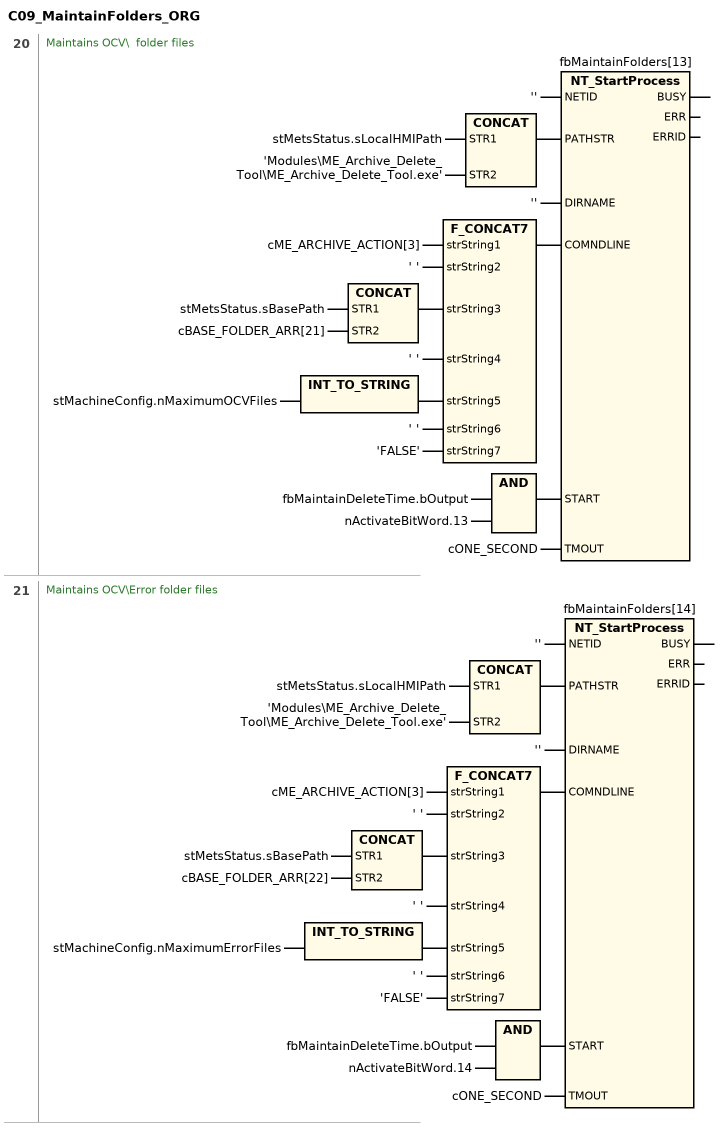
// NETWORK 20
// Maintains OCV\  folder files
fbMaintainFolders[13](
    NETID := '',
    PATHSTR := CONCAT(STR1 := stMetsStatus.sLocalHMIPath, STR2 := 'Modules\ME_Archive_Delete_Tool\ME_Archive_Delete_Tool.exe'),
    DIRNAME := '',
    COMNDLINE := F_CONCAT7(strString1 := cME_ARCHIVE_ACTION[3], strString2 := ' ', strString3 := CONCAT(STR1 := stMetsStatus.sBasePath, STR2 := cBASE_FOLDER_ARR[21]), strString4 := ' ', strString5 := INT_TO_STRING(stMachineConfig.nMaximumOCVFiles), strString6 := ' ', strString7 := 'FALSE'),
    START := fbMaintainDeleteTime.bOutput AND nActivateBitWord.13,
    TMOUT := cONE_SECOND); // NT_StartProcess

// NETWORK 21
// Maintains OCV\Error folder files
fbMaintainFolders[14](
    NETID := '',
    PATHSTR := CONCAT(STR1 := stMetsStatus.sLocalHMIPath, STR2 := 'Modules\ME_Archive_Delete_Tool\ME_Archive_Delete_Tool.exe'),
    DIRNAME := '',
    COMNDLINE := F_CONCAT7(strString1 := cME_ARCHIVE_ACTION[3], strString2 := ' ', strString3 := CONCAT(STR1 := stMetsStatus.sBasePath, STR2 := cBASE_FOLDER_ARR[22]), strString4 := ' ', strString5 := INT_TO_STRING(stMachineConfig.nMaximumErrorFiles), strString6 := ' ', strString7 := 'FALSE'),
    START := fbMaintainDeleteTime.bOutput AND nActivateBitWord.14,
    TMOUT := cONE_SECOND); // NT_StartProcess

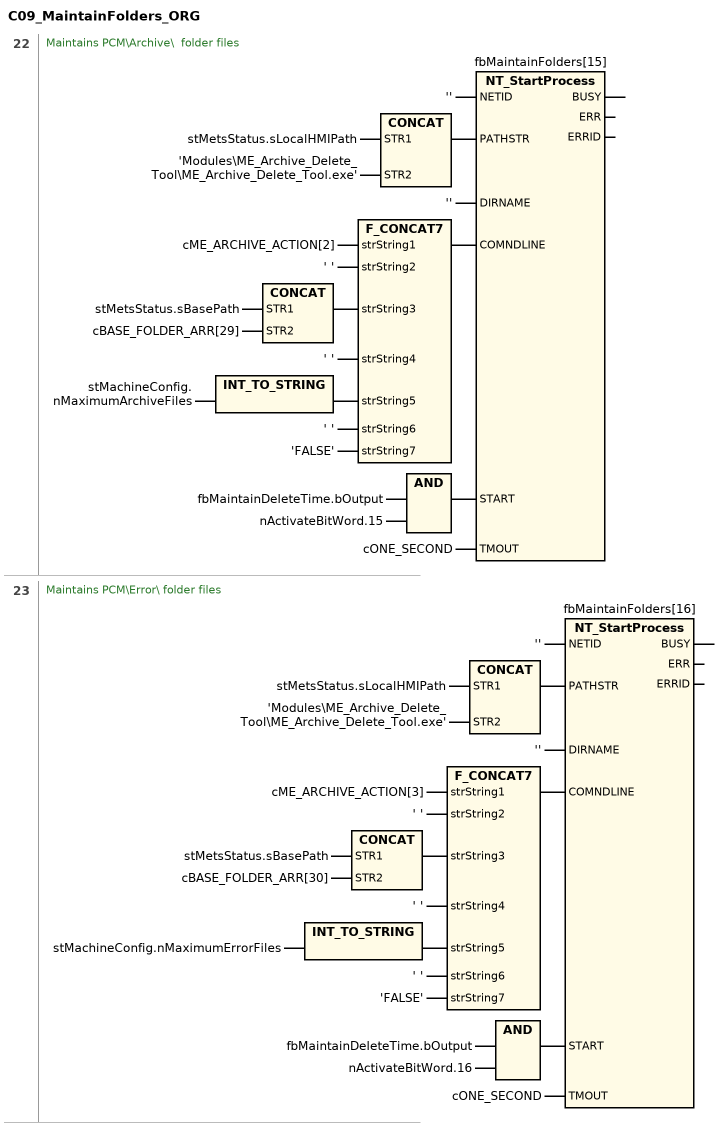
// NETWORK 22
// Maintains PCM\Archive\  folder files
fbMaintainFolders[15](
    NETID := '',
    PATHSTR := CONCAT(STR1 := stMetsStatus.sLocalHMIPath, STR2 := 'Modules\ME_Archive_Delete_Tool\ME_Archive_Delete_Tool.exe'),
    DIRNAME := '',
    COMNDLINE := F_CONCAT7(strString1 := cME_ARCHIVE_ACTION[2], strString2 := ' ', strString3 := CONCAT(STR1 := stMetsStatus.sBasePath, STR2 := cBASE_FOLDER_ARR[29]), strString4 := ' ', strString5 := INT_TO_STRING(stMachineConfig.nMaximumArchiveFiles), strString6 := ' ', strString7 := 'FALSE'),
    START := fbMaintainDeleteTime.bOutput AND nActivateBitWord.15,
    TMOUT := cONE_SECOND); // NT_StartProcess

// NETWORK 23
// Maintains PCM\Error\ folder files
fbMaintainFolders[16](
    NETID := '',
    PATHSTR := CONCAT(STR1 := stMetsStatus.sLocalHMIPath, STR2 := 'Modules\ME_Archive_Delete_Tool\ME_Archive_Delete_Tool.exe'),
    DIRNAME := '',
    COMNDLINE := F_CONCAT7(strString1 := cME_ARCHIVE_ACTION[3], strString2 := ' ', strString3 := CONCAT(STR1 := stMetsStatus.sBasePath, STR2 := cBASE_FOLDER_ARR[30]), strString4 := ' ', strString5 := INT_TO_STRING(stMachineConfig.nMaximumErrorFiles), strString6 := ' ', strString7 := 'FALSE'),
    START := fbMaintainDeleteTime.bOutput AND nActivateBitWord.16,
    TMOUT := cONE_SECOND); // NT_StartProcess

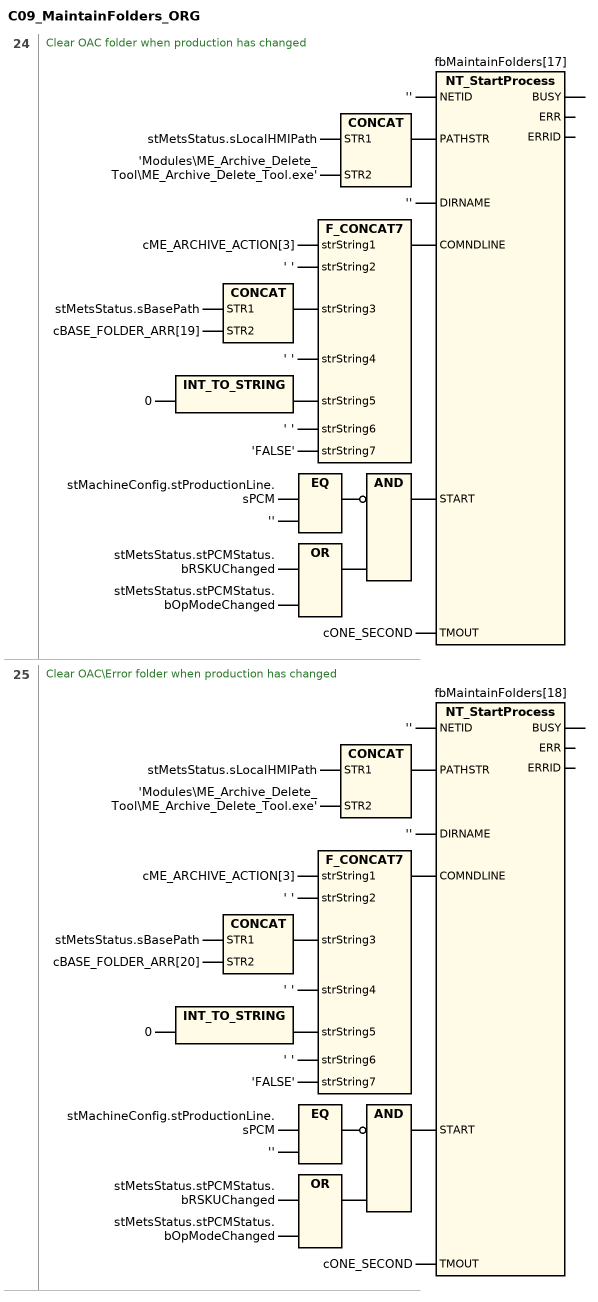
// NETWORK 24
// Clear OAC folder when production has changed
fbMaintainFolders[17](
    NETID := '',
    PATHSTR := CONCAT(STR1 := stMetsStatus.sLocalHMIPath, STR2 := 'Modules\ME_Archive_Delete_Tool\ME_Archive_Delete_Tool.exe'),
    DIRNAME := '',
    COMNDLINE := F_CONCAT7(strString1 := cME_ARCHIVE_ACTION[3], strString2 := ' ', strString3 := CONCAT(STR1 := stMetsStatus.sBasePath, STR2 := cBASE_FOLDER_ARR[19]), strString4 := ' ', strString5 := INT_TO_STRING(0), strString6 := ' ', strString7 := 'FALSE'),
    START := NOT (stMachineConfig.stProductionLine.sPCM = '') AND (stMetsStatus.stPCMStatus.bRSKUChanged OR stMetsStatus.stPCMStatus.bOpModeChanged),
    TMOUT := cONE_SECOND); // NT_StartProcess

// NETWORK 25
// Clear OAC\Error folder when production has changed
fbMaintainFolders[18](
    NETID := '',
    PATHSTR := CONCAT(STR1 := stMetsStatus.sLocalHMIPath, STR2 := 'Modules\ME_Archive_Delete_Tool\ME_Archive_Delete_Tool.exe'),
    DIRNAME := '',
    COMNDLINE := F_CONCAT7(strString1 := cME_ARCHIVE_ACTION[3], strString2 := ' ', strString3 := CONCAT(STR1 := stMetsStatus.sBasePath, STR2 := cBASE_FOLDER_ARR[20]), strString4 := ' ', strString5 := INT_TO_STRING(0), strString6 := ' ', strString7 := 'FALSE'),
    START := NOT (stMachineConfig.stProductionLine.sPCM = '') AND (stMetsStatus.stPCMStatus.bRSKUChanged OR stMetsStatus.stPCMStatus.bOpModeChanged),
    TMOUT := cONE_SECOND); // NT_StartProcess

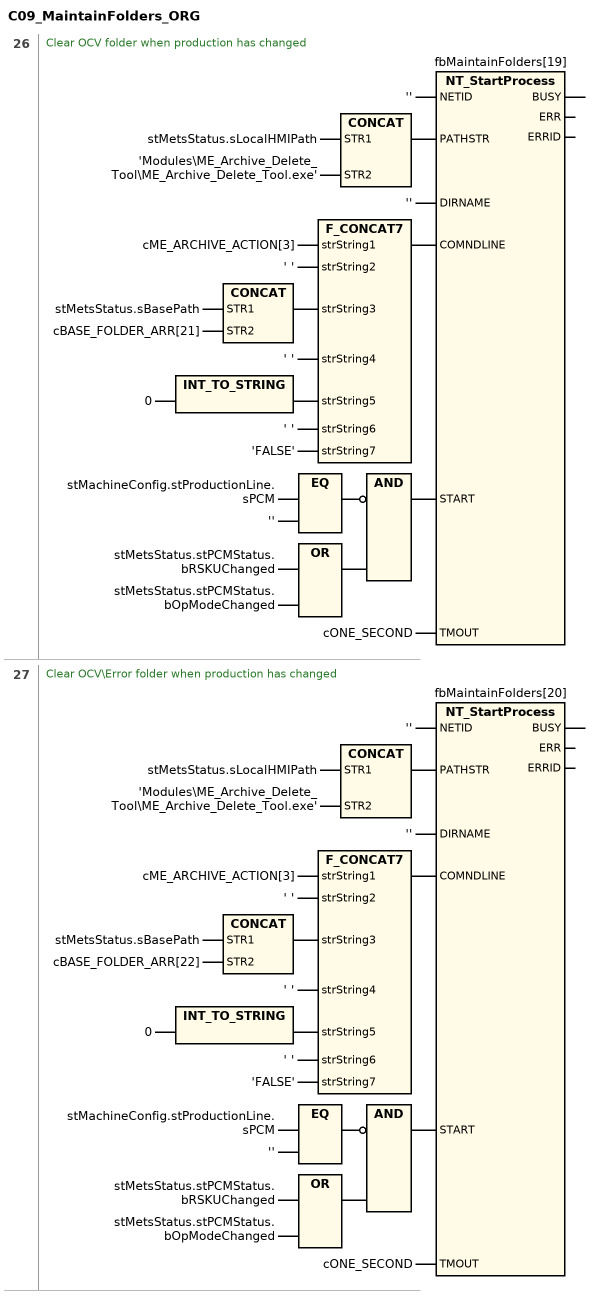
// NETWORK 26
// Clear OCV folder when production has changed
fbMaintainFolders[19](
    NETID := '',
    PATHSTR := CONCAT(STR1 := stMetsStatus.sLocalHMIPath, STR2 := 'Modules\ME_Archive_Delete_Tool\ME_Archive_Delete_Tool.exe'),
    DIRNAME := '',
    COMNDLINE := F_CONCAT7(strString1 := cME_ARCHIVE_ACTION[3], strString2 := ' ', strString3 := CONCAT(STR1 := stMetsStatus.sBasePath, STR2 := cBASE_FOLDER_ARR[21]), strString4 := ' ', strString5 := INT_TO_STRING(0), strString6 := ' ', strString7 := 'FALSE'),
    START := NOT (stMachineConfig.stProductionLine.sPCM = '') AND (stMetsStatus.stPCMStatus.bRSKUChanged OR stMetsStatus.stPCMStatus.bOpModeChanged),
    TMOUT := cONE_SECOND); // NT_StartProcess

// NETWORK 27
// Clear OCV\Error folder when production has changed
fbMaintainFolders[20](
    NETID := '',
    PATHSTR := CONCAT(STR1 := stMetsStatus.sLocalHMIPath, STR2 := 'Modules\ME_Archive_Delete_Tool\ME_Archive_Delete_Tool.exe'),
    DIRNAME := '',
    COMNDLINE := F_CONCAT7(strString1 := cME_ARCHIVE_ACTION[3], strString2 := ' ', strString3 := CONCAT(STR1 := stMetsStatus.sBasePath, STR2 := cBASE_FOLDER_ARR[22]), strString4 := ' ', strString5 := INT_TO_STRING(0), strString6 := ' ', strString7 := 'FALSE'),
    START := NOT (stMachineConfig.stProductionLine.sPCM = '') AND (stMetsStatus.stPCMStatus.bRSKUChanged OR stMetsStatus.stPCMStatus.bOpModeChanged),
    TMOUT := cONE_SECOND); // NT_StartProcess

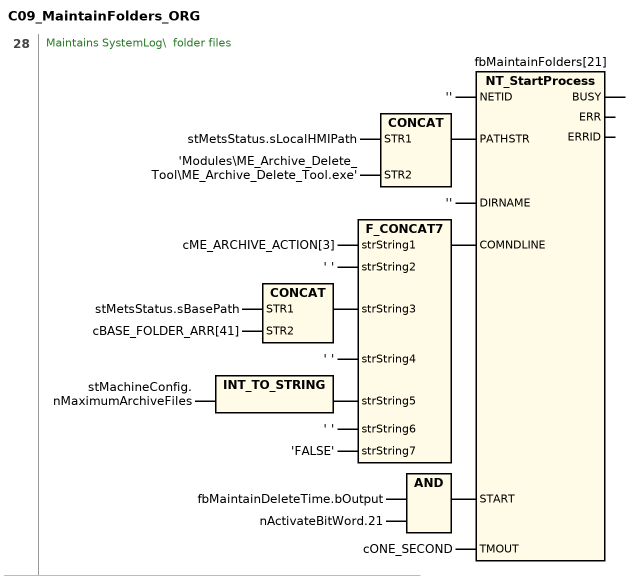
// NETWORK 28
// Maintains SystemLog\  folder files
fbMaintainFolders[21](
    NETID := '',
    PATHSTR := CONCAT(STR1 := stMetsStatus.sLocalHMIPath, STR2 := 'Modules\ME_Archive_Delete_Tool\ME_Archive_Delete_Tool.exe'),
    DIRNAME := '',
    COMNDLINE := F_CONCAT7(strString1 := cME_ARCHIVE_ACTION[3], strString2 := ' ', strString3 := CONCAT(STR1 := stMetsStatus.sBasePath, STR2 := cBASE_FOLDER_ARR[41]), strString4 := ' ', strString5 := INT_TO_STRING(stMachineConfig.nMaximumArchiveFiles), strString6 := ' ', strString7 := 'FALSE'),
    START := fbMaintainDeleteTime.bOutput AND nActivateBitWord.21,
    TMOUT := cONE_SECOND); // NT_StartProcess

ACTION ShiftActivationBit:
IF fbMaintainDeleteTime.bOutput	THEN
	IF nActivateBitWord = 0 THEN
		nActivateBitWord := 1;
	ELSE
		nActivateBitWord :=SHL(nActivateBitWord,1);
	END_IF
END_IF
END_ACTION

END_PROGRAM

// ---- POUs/_Exclude/F15_CaseControlCACData_ORG.TcPOU
PROGRAM F15_CaseControlCACData_ORG
VAR
	rtrigScanBarcode				: R_TRIG;
	fbScannerCtrl					: FB_SCANNER_CameraSelect;
	bScanCaseLabel				: BOOL;
	fbCaseLableEvaluation			: FB_SCANNER_Evaluation;

	rtrigSetCaseValidationOK			: R_TRIG;
	rtrigSetCaseValidationNOK		: R_TRIG;

	sCaseSerialCode				: T_CASE_Barcode;
	sFirstOuterInCase				: T_OUTER_Barcode;
	sLastOuterInCase				: T_OUTER_Barcode;
	sFirstPackSerialCode			: T_PACK_Barcode;
	sLastPackSerialCode				: T_PACK_Barcode;


	fbSequenceControl				: FB_SYSTEM_SeqControl;
	nSequenceStep				: INT;
	b00_Idle						: BOOL;
	b01_ScanLabel					: BOOL;
	b03_CreateFileName			: BOOL;
	b05_MoveCaseData				: BOOL;
	b08_WriteFSSFile				: BOOL;
	b10_CaseTraceValid			: BOOL;
	b18_CaseValid					: BOOL;
	b19_CaseInvalid				: BOOL;
	b20_Done						: BOOL;

	bDone						: BOOL;
	bBusy						: BOOL;
	tonScanTimeout					: TON;
	tonOverTime				: TON;

	rtrigCACData				: R_TRIG;
	tF15TimeExecution		: TIME;
	bTestSeq						: BOOL;
	sCACFileTemplate				: T_CAC_Filename;

	stValidateCACData				: ST_CAC_Data;
	fbMoveCaseData				: FB_CASE_ValidateAndMoveCACData;

	sPrintCaseContent				: STRING(255);

	fbPopulateCHMData				: FB_CHM_PopulateDataForFSS3;
	fbWriteCHMFile				: FB_CHM_WriteFSS3Files; (*Old system supporting FSS2 -> FB_CHM_WriteFSSFile;*)

	fbWriteCACToArchive 			: FB_CAC_WriteToArchive_v2;
	fbWriteCACToArchiveDB			: FB_CAC_WriteHierachyToDB;
	fbCaseStatusPulse				: TON;
	bCACValid					: BOOL;
	bCHMValid					: BOOL;


	fbMoveVerifiedCAC				: FB_CASE_MoveVerifiedCAC;
	fbMoveFailedCAC				: FB_CASE_MoveFailedCAC;

	fbCaseEfficiency				: FB_KPI_GenericEfficiency;
	fbCaseInspectionEfficiency		: FB_KPI_CaseEfficiency;
	(*fbCaseInspectionEfficiency		: FB_KPI_PACAN_CaseEfficiency;*)
	fbRejectCount					: CTU;
	nRejectActualCount				: INT;

	fbCaseValidationScanned			: FB_CTU32;
	fbCaseValidationCorrect			: FB_CTU32;
	fbCaseValidationNoCaseLabel		: FB_CTU32;
	fbCaseValidationCasePackerReject	: FB_CTU32;

	aLastCaseBarcodes				: ARRAY[1..cMAX_LAST_CASE_BARCODES] OF T_CASE_Barcode;
	fbAddVerifiedCaseBarcode		: FB_CASE_AddVerifiedCaseBarcode;

	fbCaseLevelCounter	: FB_KPI_CaseLevelCounter;
	tofCaseValidationCameraOFFDelay 	: TOF;

	fbFileWriteCACError				: FB_LOG_FileWriteError;
	fbFileWriteCHMError			: FB_LOG_FileWriteError;

END_VAR
(*
VAR CONSTANT
	sOptions						: ST_SCANNER_Options := (eScannerType := E_MV_440SR_FULL, nImageBuffer := 1, nExpectedResp := 1);
END_VAR*)
VAR // added by the converter: edge detectors and wires of the graphical bodies
    _w1 : ANY;
    _w2, _w3 : BOOL;
END_VAR

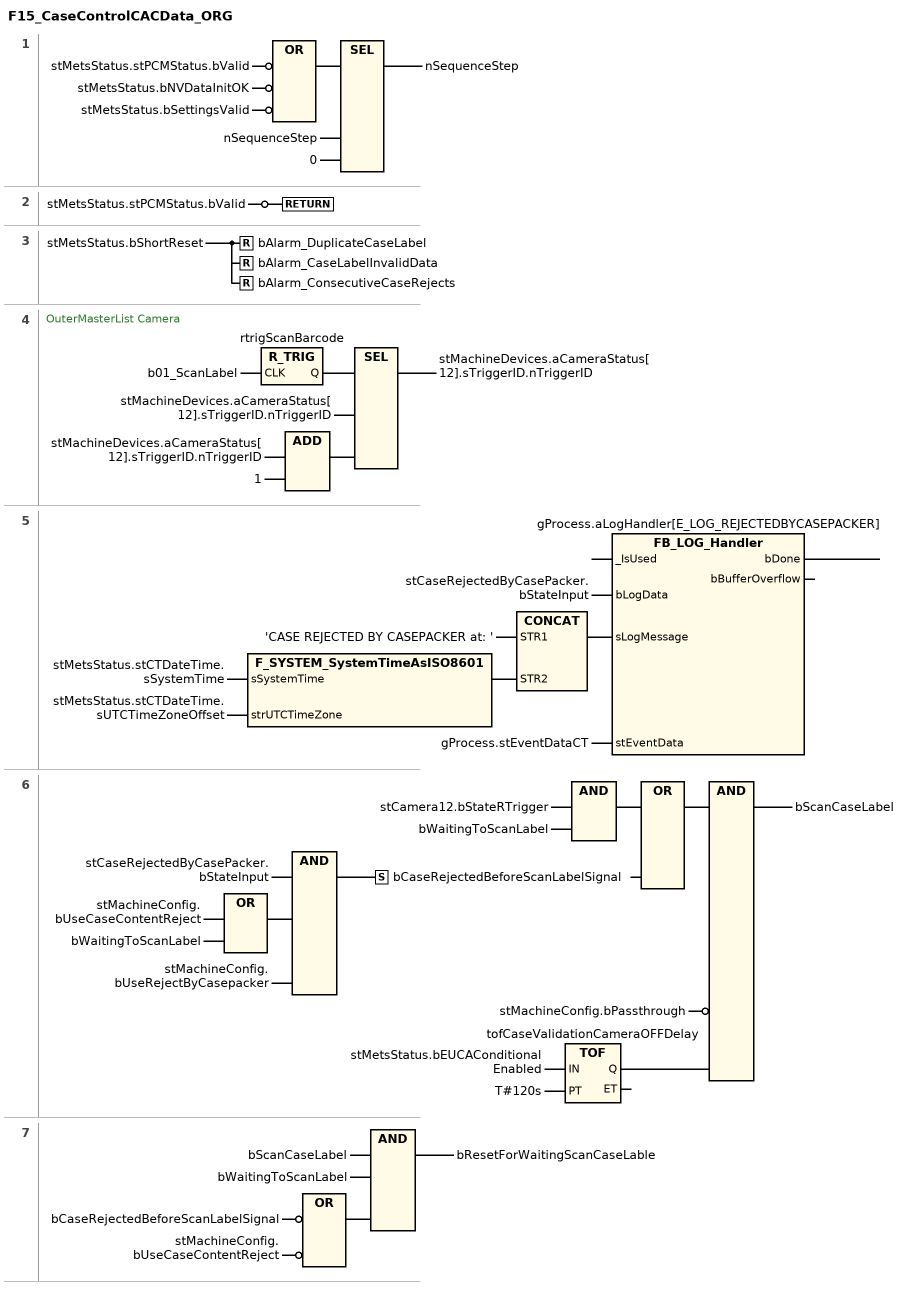
// NETWORK 1
nSequenceStep := SEL(NOT stMetsStatus.stPCMStatus.bValid OR NOT stMetsStatus.bNVDataInitOK OR NOT stMetsStatus.bSettingsValid, nSequenceStep, 0);

// NETWORK 2
IF NOT stMetsStatus.stPCMStatus.bValid THEN RETURN; END_IF

// NETWORK 3
bAlarm_DuplicateCaseLabel R= stMetsStatus.bShortReset;
bAlarm_CaseLabelInvalidData R= stMetsStatus.bShortReset;
bAlarm_ConsecutiveCaseRejects R= stMetsStatus.bShortReset;

// NETWORK 4
// OuterMasterList Camera
rtrigScanBarcode(CLK := b01_ScanLabel); // R_TRIG
stMachineDevices.aCameraStatus[12].sTriggerID.nTriggerID := SEL(rtrigScanBarcode.Q, stMachineDevices.aCameraStatus[12].sTriggerID.nTriggerID, stMachineDevices.aCameraStatus[12].sTriggerID.nTriggerID + 1);

// NETWORK 5
gProcess.aLogHandler[E_LOG_REJECTEDBYCASEPACKER](
    bLogData := stCaseRejectedByCasePacker.bStateInput,
    sLogMessage := CONCAT(STR1 := 'CASE REJECTED BY CASEPACKER at: ', STR2 := F_SYSTEM_SystemTimeAsISO8601(sSystemTime := stMetsStatus.stCTDateTime.sSystemTime, strUTCTimeZone := stMetsStatus.stCTDateTime.sUTCTimeZoneOffset)),
    stEventData := gProcess.stEventDataCT); // FB_LOG_Handler

// NETWORK 6
_w1 := stCaseRejectedByCasePacker.bStateInput AND (stMachineConfig.bUseCaseContentReject OR bWaitingToScanLabel) AND stMachineConfig.bUseRejectByCasepacker;
bCaseRejectedBeforeScanLabelSignal S= _w1;
tofCaseValidationCameraOFFDelay(IN := stMetsStatus.bEUCAConditionalEnabled, PT := T#120s); // TOF
bScanCaseLabel := (stCamera12.bStateRTrigger AND bWaitingToScanLabel OR _w1) AND NOT stMachineConfig.bPassthrough AND tofCaseValidationCameraOFFDelay.Q;

// NETWORK 7
bResetForWaitingScanCaseLable := bScanCaseLabel AND bWaitingToScanLabel AND (NOT bCaseRejectedBeforeScanLabelSignal OR NOT stMachineConfig.bUseCaseContentReject);

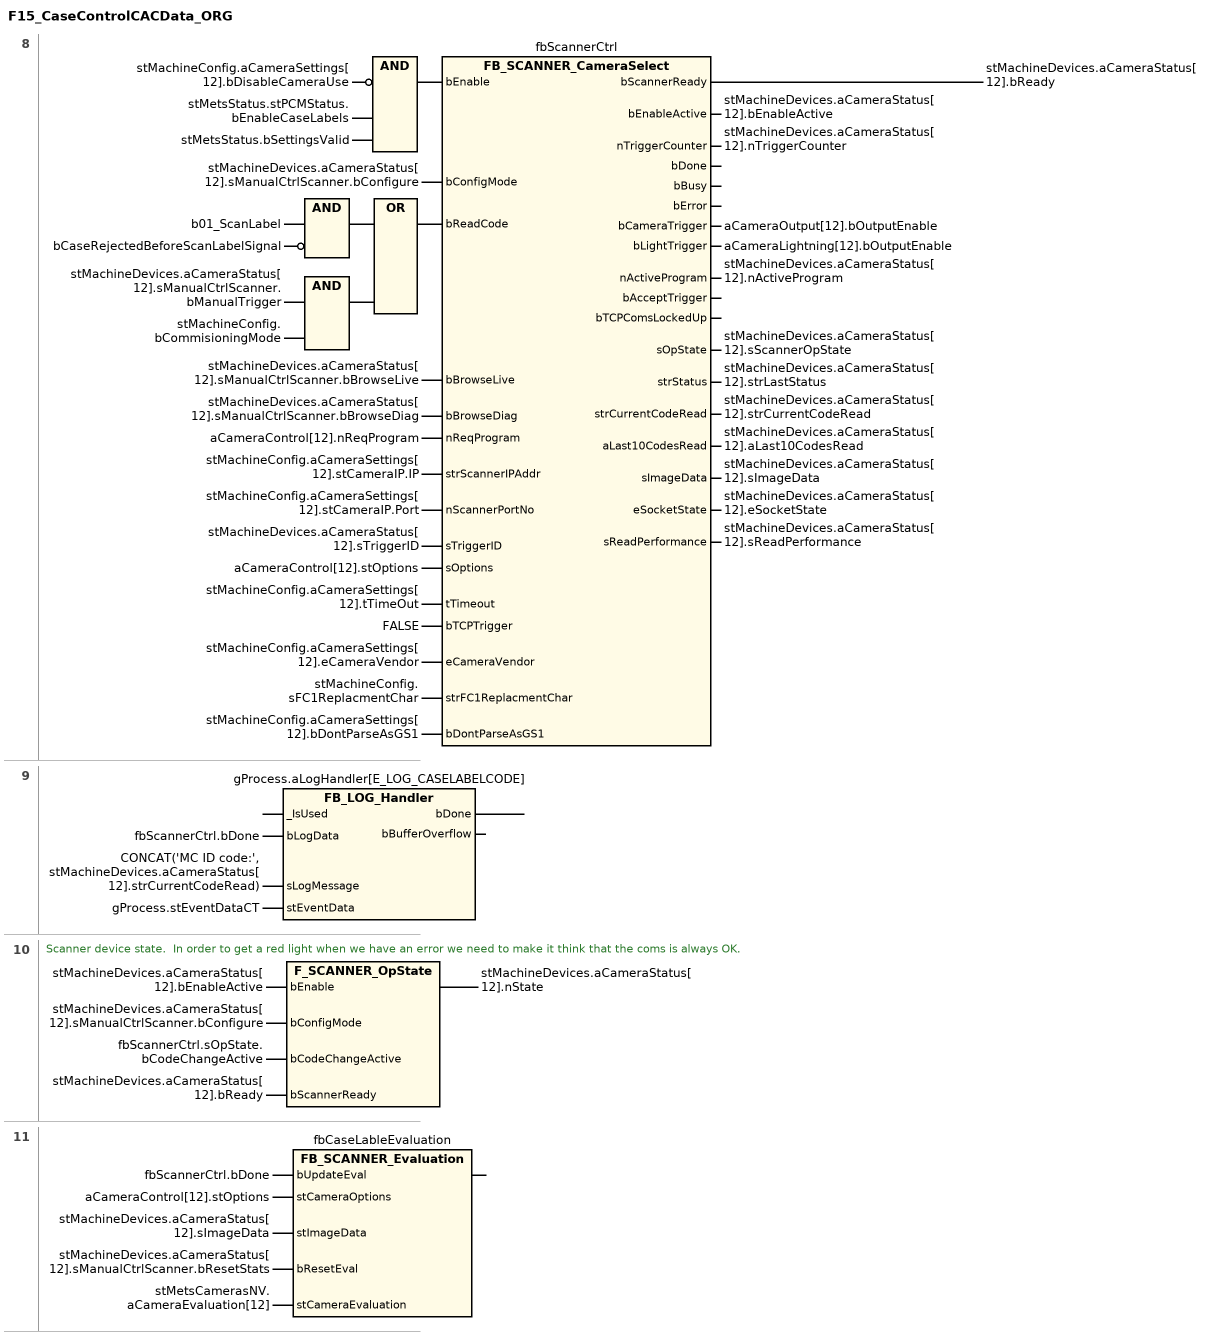
// NETWORK 8
fbScannerCtrl(
    bEnable := NOT stMachineConfig.aCameraSettings[12].bDisableCameraUse AND stMetsStatus.stPCMStatus.bEnableCaseLabels AND stMetsStatus.bSettingsValid,
    bConfigMode := stMachineDevices.aCameraStatus[12].sManualCtrlScanner.bConfigure,
    bReadCode := b01_ScanLabel AND NOT bCaseRejectedBeforeScanLabelSignal OR stMachineDevices.aCameraStatus[12].sManualCtrlScanner.bManualTrigger AND stMachineConfig.bCommisioningMode,
    bBrowseLive := stMachineDevices.aCameraStatus[12].sManualCtrlScanner.bBrowseLive,
    bBrowseDiag := stMachineDevices.aCameraStatus[12].sManualCtrlScanner.bBrowseDiag,
    nReqProgram := aCameraControl[12].nReqProgram,
    strScannerIPAddr := stMachineConfig.aCameraSettings[12].stCameraIP.IP,
    nScannerPortNo := stMachineConfig.aCameraSettings[12].stCameraIP.Port,
    sTriggerID := stMachineDevices.aCameraStatus[12].sTriggerID,
    sOptions := aCameraControl[12].stOptions,
    tTimeout := stMachineConfig.aCameraSettings[12].tTimeOut,
    bTCPTrigger := FALSE,
    eCameraVendor := stMachineConfig.aCameraSettings[12].eCameraVendor,
    strFC1ReplacmentChar := stMachineConfig.sFC1ReplacmentChar,
    bDontParseAsGS1 := stMachineConfig.aCameraSettings[12].bDontParseAsGS1,
    bEnableActive => stMachineDevices.aCameraStatus[12].bEnableActive,
    nTriggerCounter => stMachineDevices.aCameraStatus[12].nTriggerCounter,
    bCameraTrigger => aCameraOutput[12].bOutputEnable,
    bLightTrigger => aCameraLightning[12].bOutputEnable,
    nActiveProgram => stMachineDevices.aCameraStatus[12].nActiveProgram,
    sOpState => stMachineDevices.aCameraStatus[12].sScannerOpState,
    strStatus => stMachineDevices.aCameraStatus[12].strLastStatus,
    strCurrentCodeRead => stMachineDevices.aCameraStatus[12].strCurrentCodeRead,
    aLast10CodesRead => stMachineDevices.aCameraStatus[12].aLast10CodesRead,
    sImageData => stMachineDevices.aCameraStatus[12].sImageData,
    eSocketState => stMachineDevices.aCameraStatus[12].eSocketState,
    sReadPerformance => stMachineDevices.aCameraStatus[12].sReadPerformance); // FB_SCANNER_CameraSelect
stMachineDevices.aCameraStatus[12].bReady := fbScannerCtrl.bScannerReady;

// NETWORK 9
gProcess.aLogHandler[E_LOG_CASELABELCODE](
    bLogData := fbScannerCtrl.bDone,
    sLogMessage := CONCAT('MC ID code:', stMachineDevices.aCameraStatus[12].strCurrentCodeRead),
    stEventData := gProcess.stEventDataCT); // FB_LOG_Handler

// NETWORK 10
// Scanner device state.  In order to get a red light when we have an error we need to make it think that the coms is always OK.
stMachineDevices.aCameraStatus[12].nState := F_SCANNER_OpState(bEnable := stMachineDevices.aCameraStatus[12].bEnableActive, bConfigMode := stMachineDevices.aCameraStatus[12].sManualCtrlScanner.bConfigure, bCodeChangeActive := fbScannerCtrl.sOpState.bCodeChangeActive, bScannerReady := stMachineDevices.aCameraStatus[12].bReady);

// NETWORK 11
fbCaseLableEvaluation(
    bUpdateEval := fbScannerCtrl.bDone,
    stCameraOptions := aCameraControl[12].stOptions,
    stImageData := stMachineDevices.aCameraStatus[12].sImageData,
    bResetEval := stMachineDevices.aCameraStatus[12].sManualCtrlScanner.bResetStats,
    stCameraEvaluation := stMetsCamerasNV.aCameraEvaluation[12]); // FB_SCANNER_Evaluation

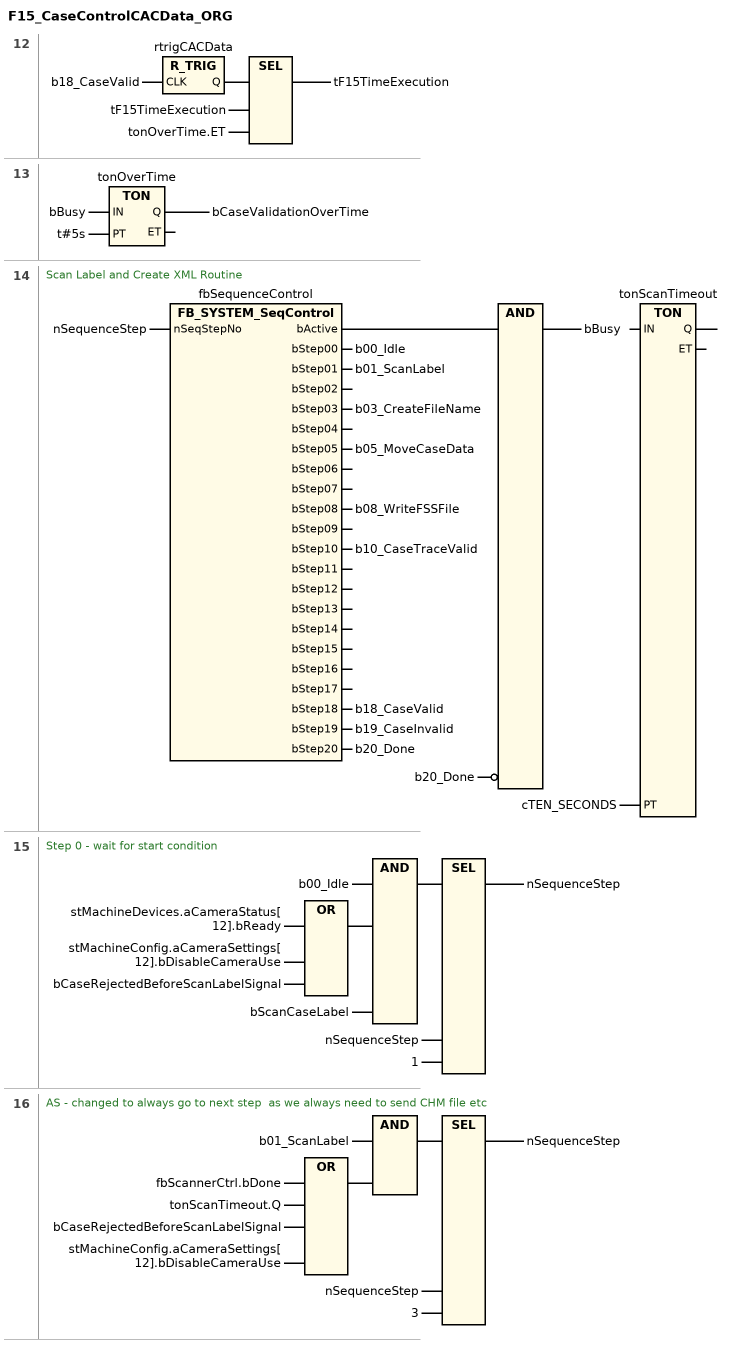
// NETWORK 12
rtrigCACData(CLK := b18_CaseValid); // R_TRIG
tF15TimeExecution := SEL(rtrigCACData.Q, tF15TimeExecution, tonOverTime.ET);

// NETWORK 13
tonOverTime(IN := bBusy, PT := t#5s); // TON
bCaseValidationOverTime := tonOverTime.Q;

// NETWORK 14
// 					Scan Label and Create XML Routine
//
//
//
fbSequenceControl(
    nSeqStepNo := nSequenceStep,
    bStep00 => b00_Idle,
    bStep01 => b01_ScanLabel,
    bStep03 => b03_CreateFileName,
    bStep05 => b05_MoveCaseData,
    bStep08 => b08_WriteFSSFile,
    bStep10 => b10_CaseTraceValid,
    bStep18 => b18_CaseValid,
    bStep19 => b19_CaseInvalid,
    bStep20 => b20_Done); // FB_SYSTEM_SeqControl
_w2 := fbSequenceControl.bActive AND NOT b20_Done;
bBusy := _w2;
tonScanTimeout(IN := _w2, PT := cTEN_SECONDS); // TON

// NETWORK 15
// 					Step 0 - wait for start condition
//
//
nSequenceStep := SEL(b00_Idle AND (stMachineDevices.aCameraStatus[12].bReady OR stMachineConfig.aCameraSettings[12].bDisableCameraUse OR bCaseRejectedBeforeScanLabelSignal) AND bScanCaseLabel, nSequenceStep, 1);

// NETWORK 16
// 					AS - changed to always go to next step  as we always need to send CHM file etc
//
//
nSequenceStep := SEL(b01_ScanLabel AND (fbScannerCtrl.bDone OR tonScanTimeout.Q OR bCaseRejectedBeforeScanLabelSignal OR stMachineConfig.aCameraSettings[12].bDisableCameraUse), nSequenceStep, 3);

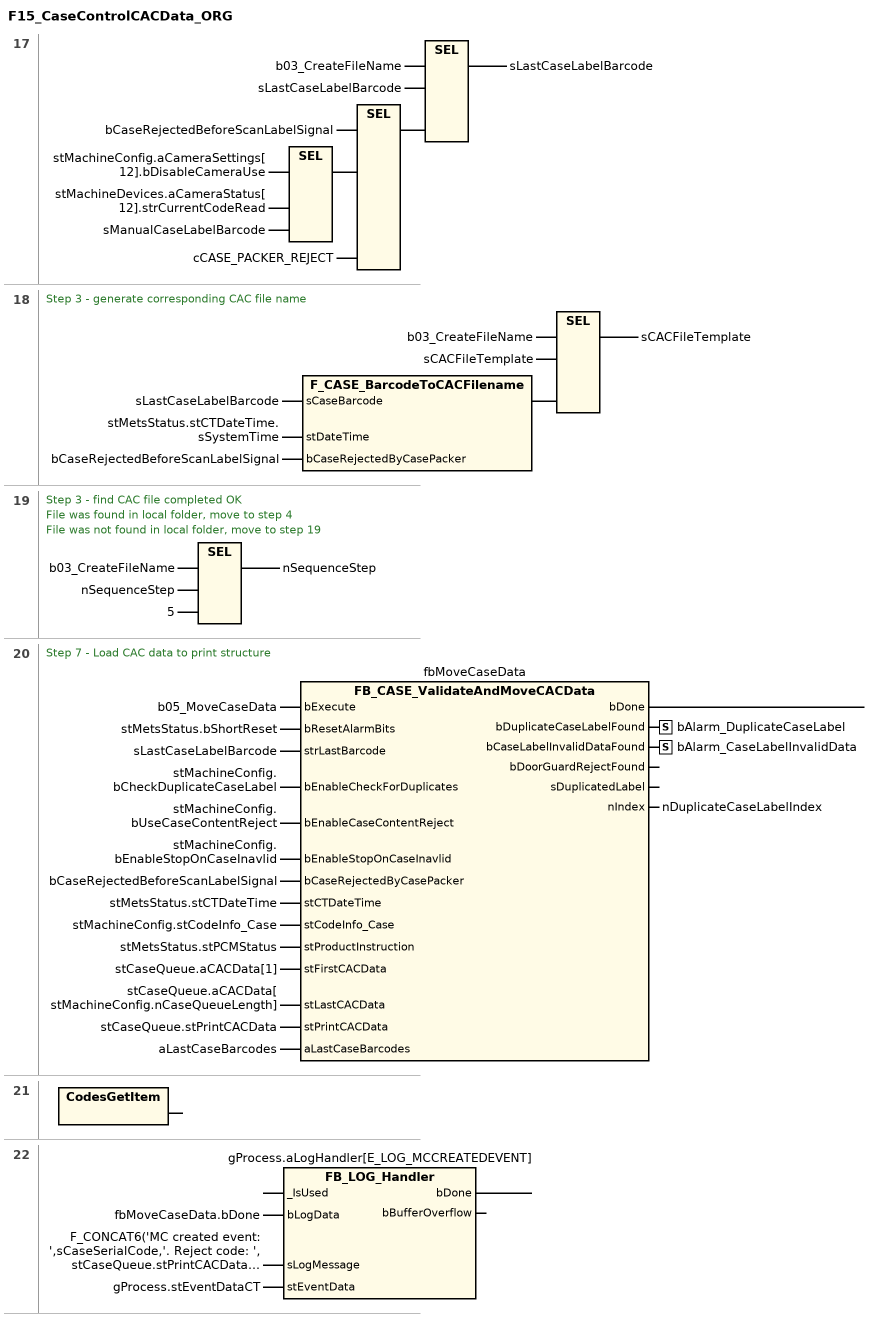
// NETWORK 17
sLastCaseLabelBarcode := SEL(b03_CreateFileName, sLastCaseLabelBarcode, SEL(bCaseRejectedBeforeScanLabelSignal, SEL(stMachineConfig.aCameraSettings[12].bDisableCameraUse, stMachineDevices.aCameraStatus[12].strCurrentCodeRead, sManualCaseLabelBarcode), cCASE_PACKER_REJECT));

// NETWORK 18
// Step 3 - generate corresponding CAC file name
sCACFileTemplate := SEL(b03_CreateFileName, sCACFileTemplate, F_CASE_BarcodeToCACFilename(sCaseBarcode := sLastCaseLabelBarcode, stDateTime := stMetsStatus.stCTDateTime.sSystemTime, bCaseRejectedByCasePacker := bCaseRejectedBeforeScanLabelSignal));

// NETWORK 19
// 					Step 3 - find CAC file completed OK
// File was found in local folder, move to step 4
// File was not found in local folder, move to step 19
//
nSequenceStep := SEL(b03_CreateFileName, nSequenceStep, 5);

// NETWORK 20
// Step 7 - Load CAC data to print structure
fbMoveCaseData(
    bExecute := b05_MoveCaseData,
    bResetAlarmBits := stMetsStatus.bShortReset,
    strLastBarcode := sLastCaseLabelBarcode,
    bEnableCheckForDuplicates := stMachineConfig.bCheckDuplicateCaseLabel,
    bEnableCaseContentReject := stMachineConfig.bUseCaseContentReject,
    bEnableStopOnCaseInavlid := stMachineConfig.bEnableStopOnCaseInavlid,
    bCaseRejectedByCasePacker := bCaseRejectedBeforeScanLabelSignal,
    stCTDateTime := stMetsStatus.stCTDateTime,
    stCodeInfo_Case := stMachineConfig.stCodeInfo_Case,
    stProductInstruction := stMetsStatus.stPCMStatus,
    stFirstCACData := stCaseQueue.aCACData[1],
    stLastCACData := stCaseQueue.aCACData[stMachineConfig.nCaseQueueLength],
    stPrintCACData := stCaseQueue.stPrintCACData,
    aLastCaseBarcodes := aLastCaseBarcodes,
    nIndex => nDuplicateCaseLabelIndex); // FB_CASE_ValidateAndMoveCACData
bAlarm_DuplicateCaseLabel S= fbMoveCaseData.bDuplicateCaseLabelFound;
bAlarm_CaseLabelInvalidData S= fbMoveCaseData.bCaseLabelInvalidDataFound;

// NETWORK 21
CodesGetItem();

// NETWORK 22
gProcess.aLogHandler[E_LOG_MCCREATEDEVENT](
    bLogData := fbMoveCaseData.bDone,
    sLogMessage := F_CONCAT6('MC created event: ',sCaseSerialCode,'. Reject code: ', stCaseQueue.stPrintCACData.CaseRejectCode,', with case content: ', sPrintCaseContent),
    stEventData := gProcess.stEventDataCT); // FB_LOG_Handler

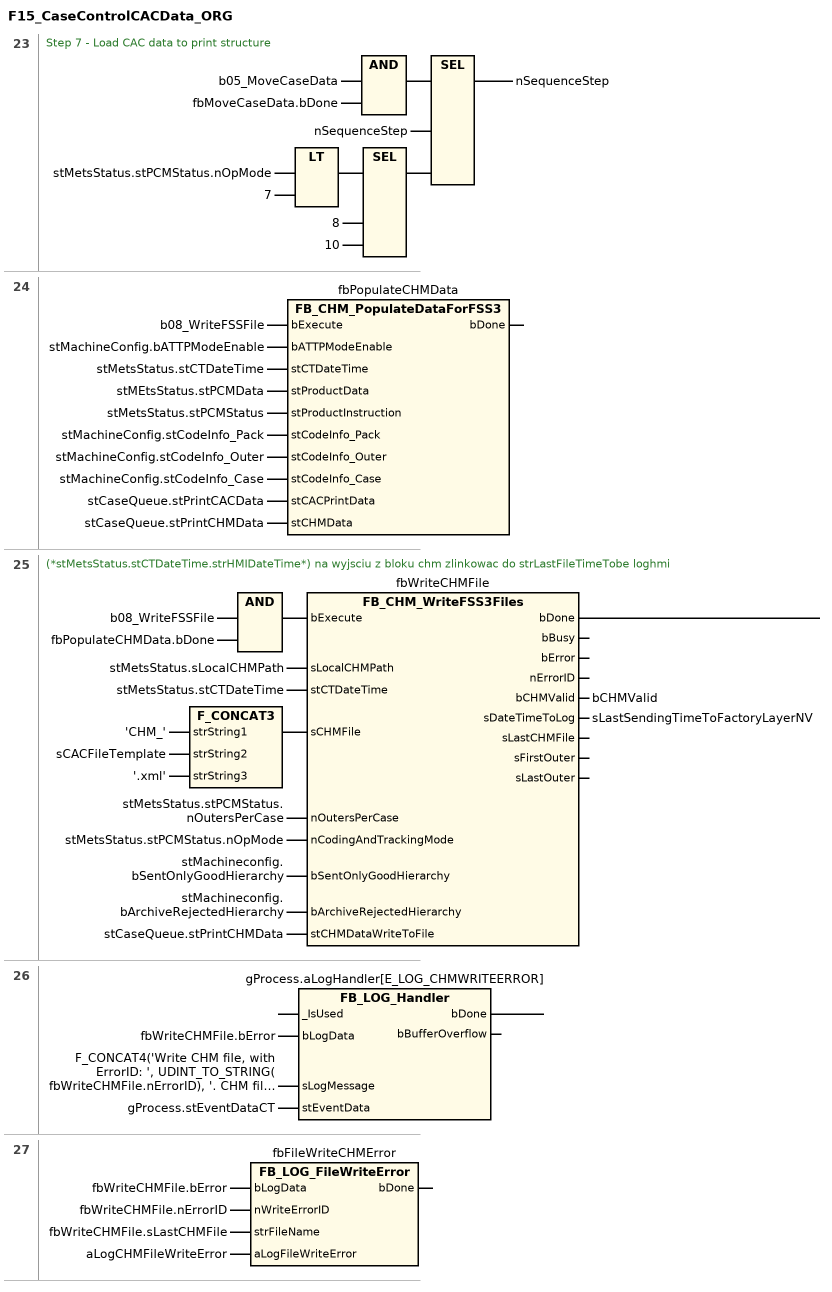
// NETWORK 23
// 					Step 7 - Load CAC data to print structure
//
//
nSequenceStep := SEL(b05_MoveCaseData AND fbMoveCaseData.bDone, nSequenceStep, SEL(stMetsStatus.stPCMStatus.nOpMode < 7, 8, 10));

// NETWORK 24
fbPopulateCHMData(
    bExecute := b08_WriteFSSFile,
    bATTPModeEnable := stMachineConfig.bATTPModeEnable,
    stCTDateTime := stMetsStatus.stCTDateTime,
    stProductData := stMEtsStatus.stPCMData,
    stProductInstruction := stMetsStatus.stPCMStatus,
    stCodeInfo_Pack := stMachineConfig.stCodeInfo_Pack,
    stCodeInfo_Outer := stMachineConfig.stCodeInfo_Outer,
    stCodeInfo_Case := stMachineConfig.stCodeInfo_Case,
    stCACPrintData := stCaseQueue.stPrintCACData,
    stCHMData := stCaseQueue.stPrintCHMData); // FB_CHM_PopulateDataForFSS3

// NETWORK 25
// (*stMetsStatus.stCTDateTime.strHMIDateTime*) na wyjsciu z bloku chm zlinkowac do strLastFileTimeTobe loghmi
fbWriteCHMFile(
    bExecute := b08_WriteFSSFile AND fbPopulateCHMData.bDone,
    sLocalCHMPath := stMetsStatus.sLocalCHMPath,
    stCTDateTime := stMetsStatus.stCTDateTime,
    sCHMFile := F_CONCAT3(strString1 := 'CHM_', strString2 := sCACFileTemplate, strString3 := '.xml'),
    nOutersPerCase := stMetsStatus.stPCMStatus.nOutersPerCase,
    nCodingAndTrackingMode := stMetsStatus.stPCMStatus.nOpMode,
    bSentOnlyGoodHierarchy := stMachineconfig.bSentOnlyGoodHierarchy,
    bArchiveRejectedHierarchy := stMachineconfig.bArchiveRejectedHierarchy,
    stCHMDataWriteToFile := stCaseQueue.stPrintCHMData,
    bCHMValid => bCHMValid,
    sDateTimeToLog => sLastSendingTimeToFactoryLayerNV); // FB_CHM_WriteFSS3Files

// NETWORK 26
gProcess.aLogHandler[E_LOG_CHMWRITEERROR](
    bLogData := fbWriteCHMFile.bError,
    sLogMessage := F_CONCAT4('Write CHM file, with ErrorID: ', UDINT_TO_STRING(fbWriteCHMFile.nErrorID), '. CHM file name: ', fbWriteCHMFile.sCHMFile),
    stEventData := gProcess.stEventDataCT); // FB_LOG_Handler

// NETWORK 27
fbFileWriteCHMError(
    bLogData := fbWriteCHMFile.bError,
    nWriteErrorID := fbWriteCHMFile.nErrorID,
    strFileName := fbWriteCHMFile.sLastCHMFile,
    aLogFileWriteError := aLogCHMFileWriteError); // FB_LOG_FileWriteError

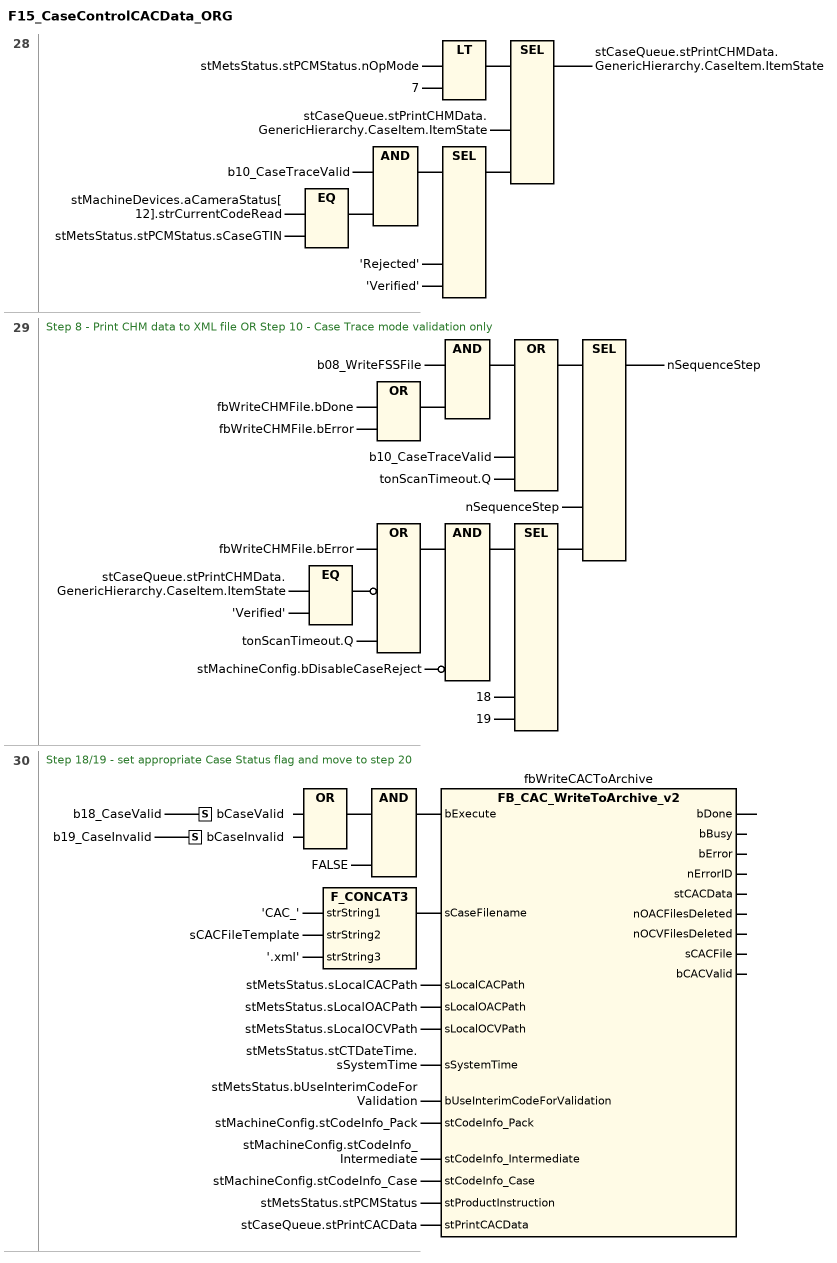
// NETWORK 28
stCaseQueue.stPrintCHMData.GenericHierarchy.CaseItem.ItemState := SEL(stMetsStatus.stPCMStatus.nOpMode < 7, stCaseQueue.stPrintCHMData.GenericHierarchy.CaseItem.ItemState, SEL(b10_CaseTraceValid AND stMachineDevices.aCameraStatus[12].strCurrentCodeRead = stMetsStatus.stPCMStatus.sCaseGTIN, 'Rejected', 'Verified'));

// NETWORK 29
// Step 8 - Print CHM data to XML file OR Step 10 - Case Trace mode validation only
nSequenceStep := SEL(b08_WriteFSSFile AND (fbWriteCHMFile.bDone OR fbWriteCHMFile.bError) OR b10_CaseTraceValid OR tonScanTimeout.Q, nSequenceStep, SEL((fbWriteCHMFile.bError OR NOT (stCaseQueue.stPrintCHMData.GenericHierarchy.CaseItem.ItemState = 'Verified') OR tonScanTimeout.Q) AND NOT stMachineConfig.bDisableCaseReject, 18, 19));

// NETWORK 30
// Step 18/19 - set appropriate Case Status flag and move to step 20
bCaseValid S= b18_CaseValid;
bCaseInvalid S= b19_CaseInvalid;
fbWriteCACToArchive(
    bExecute := (b18_CaseValid OR b19_CaseInvalid) AND FALSE,
    sCaseFilename := F_CONCAT3(strString1 := 'CAC_', strString2 := sCACFileTemplate, strString3 := '.xml'),
    sLocalCACPath := stMetsStatus.sLocalCACPath,
    sLocalOACPath := stMetsStatus.sLocalOACPath,
    sLocalOCVPath := stMetsStatus.sLocalOCVPath,
    sSystemTime := stMetsStatus.stCTDateTime.sSystemTime,
    bUseInterimCodeForValidation := stMetsStatus.bUseInterimCodeForValidation,
    stCodeInfo_Pack := stMachineConfig.stCodeInfo_Pack,
    stCodeInfo_Intermediate := stMachineConfig.stCodeInfo_Intermediate,
    stCodeInfo_Case := stMachineConfig.stCodeInfo_Case,
    stProductInstruction := stMetsStatus.stPCMStatus,
    stPrintCACData := stCaseQueue.stPrintCACData); // FB_CAC_WriteToArchive_v2

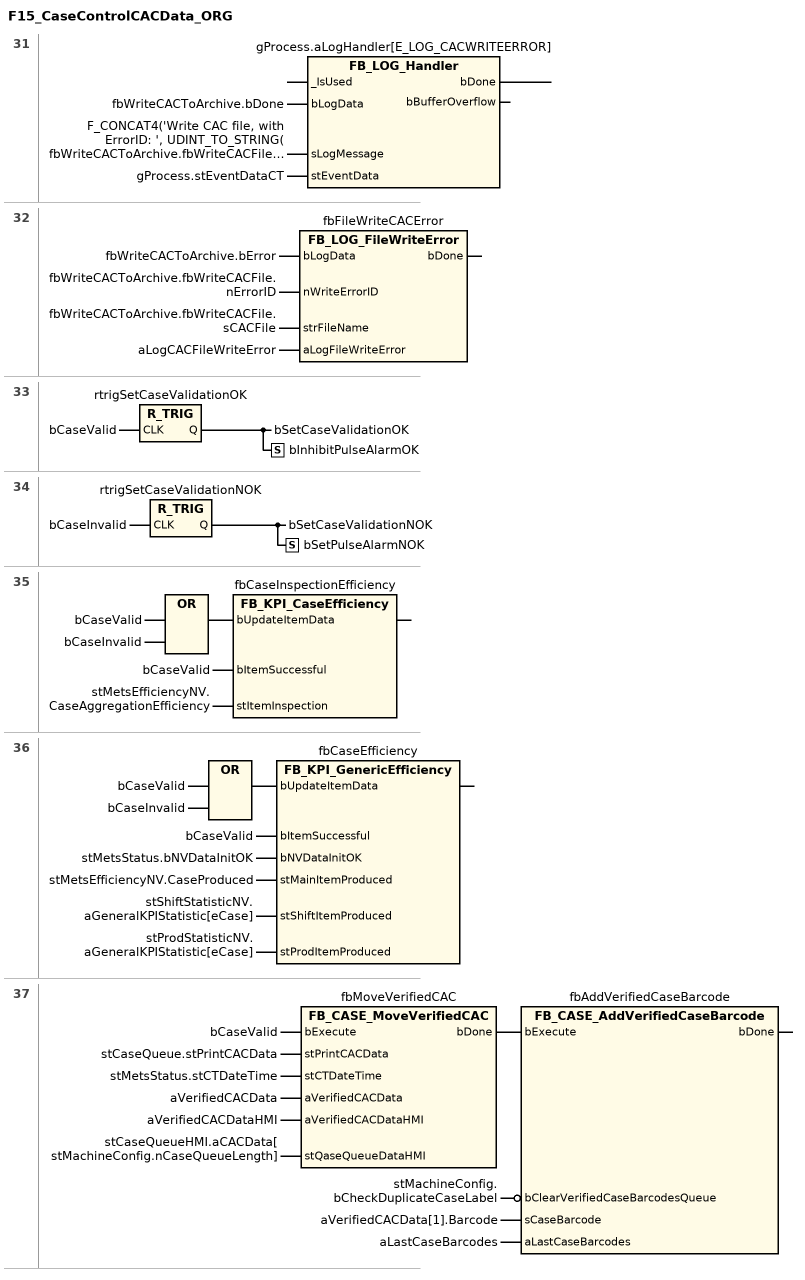
// NETWORK 31
gProcess.aLogHandler[E_LOG_CACWRITEERROR](
    bLogData := fbWriteCACToArchive.bDone,
    sLogMessage := F_CONCAT4('Write CAC file, with ErrorID: ', UDINT_TO_STRING(fbWriteCACToArchive.fbWriteCACFile.nErrorID), '. CAC file name: ', fbWriteCACToArchive.fbWriteCACFile.sCACFile),
    stEventData := gProcess.stEventDataCT); // FB_LOG_Handler

// NETWORK 32
fbFileWriteCACError(
    bLogData := fbWriteCACToArchive.bError,
    nWriteErrorID := fbWriteCACToArchive.fbWriteCACFile.nErrorID,
    strFileName := fbWriteCACToArchive.fbWriteCACFile.sCACFile,
    aLogFileWriteError := aLogCACFileWriteError); // FB_LOG_FileWriteError

// NETWORK 33
rtrigSetCaseValidationOK(CLK := bCaseValid); // R_TRIG
bSetCaseValidationOK := rtrigSetCaseValidationOK.Q;
bInhibitPulseAlarmOK S= rtrigSetCaseValidationOK.Q;

// NETWORK 34
rtrigSetCaseValidationNOK(CLK := bCaseInvalid); // R_TRIG
bSetCaseValidationNOK := rtrigSetCaseValidationNOK.Q;
bSetPulseAlarmNOK S= rtrigSetCaseValidationNOK.Q;

// NETWORK 35
fbCaseInspectionEfficiency(
    bUpdateItemData := bCaseValid OR bCaseInvalid,
    bItemSuccessful := bCaseValid,
    stItemInspection := stMetsEfficiencyNV.CaseAggregationEfficiency); // FB_KPI_CaseEfficiency

// NETWORK 36
fbCaseEfficiency(
    bUpdateItemData := bCaseValid OR bCaseInvalid,
    bItemSuccessful := bCaseValid,
    bNVDataInitOK := stMetsStatus.bNVDataInitOK,
    stMainItemProduced := stMetsEfficiencyNV.CaseProduced,
    stShiftItemProduced := stShiftStatisticNV.aGeneralKPIStatistic[eCase],
    stProdItemProduced := stProdStatisticNV.aGeneralKPIStatistic[eCase]); // FB_KPI_GenericEfficiency

// NETWORK 37
fbMoveVerifiedCAC(
    bExecute := bCaseValid,
    stPrintCACData := stCaseQueue.stPrintCACData,
    stCTDateTime := stMetsStatus.stCTDateTime,
    aVerifiedCACData := aVerifiedCACData,
    aVerifiedCACDataHMI := aVerifiedCACDataHMI,
    stQaseQueueDataHMI := stCaseQueueHMI.aCACData[stMachineConfig.nCaseQueueLength]); // FB_CASE_MoveVerifiedCAC
fbAddVerifiedCaseBarcode(
    bExecute := fbMoveVerifiedCAC.bDone,
    bClearVerifiedCaseBarcodesQueue := NOT stMachineConfig.bCheckDuplicateCaseLabel,
    sCaseBarcode := aVerifiedCACData[1].Barcode,
    aLastCaseBarcodes := aLastCaseBarcodes); // FB_CASE_AddVerifiedCaseBarcode

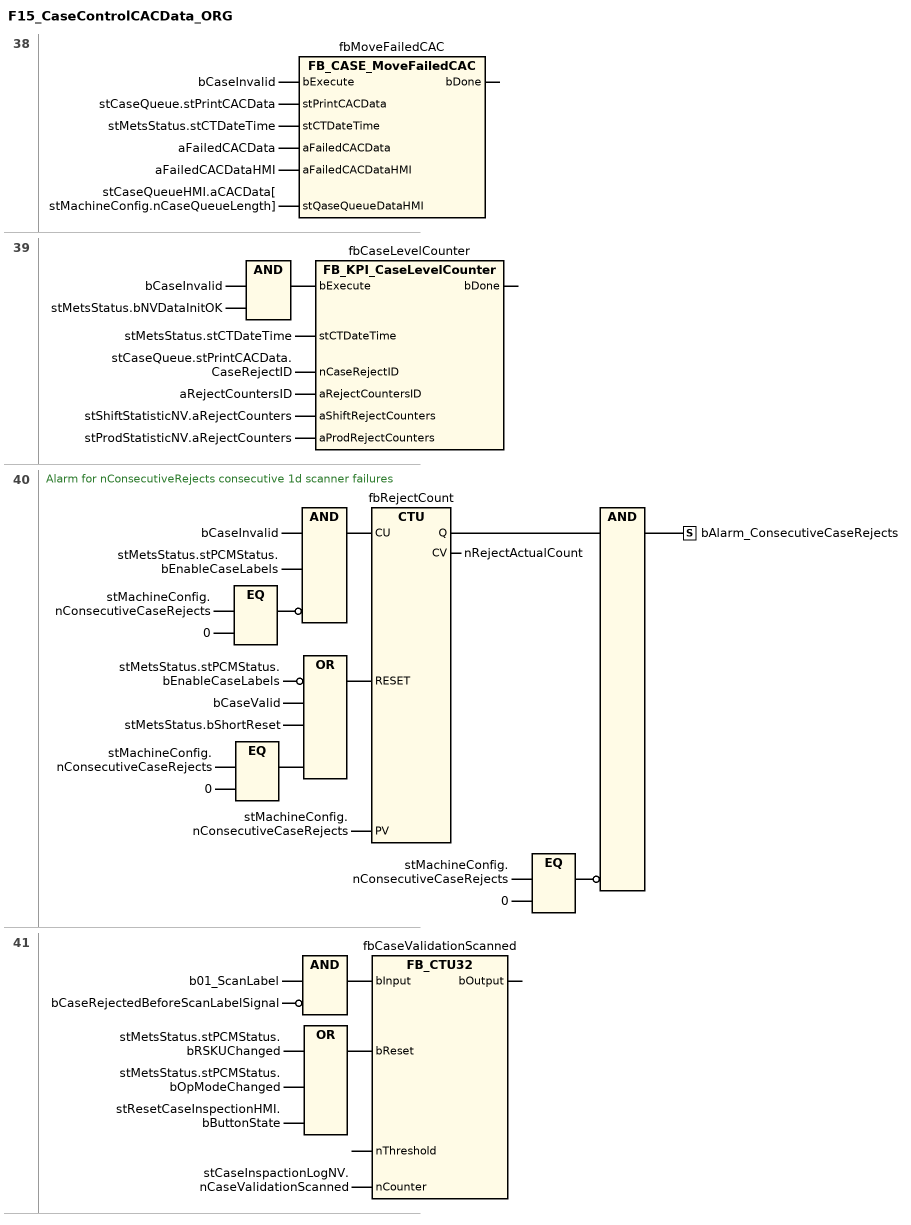
// NETWORK 38
fbMoveFailedCAC(
    bExecute := bCaseInvalid,
    stPrintCACData := stCaseQueue.stPrintCACData,
    stCTDateTime := stMetsStatus.stCTDateTime,
    aFailedCACData := aFailedCACData,
    aFailedCACDataHMI := aFailedCACDataHMI,
    stQaseQueueDataHMI := stCaseQueueHMI.aCACData[stMachineConfig.nCaseQueueLength]); // FB_CASE_MoveFailedCAC

// NETWORK 39
fbCaseLevelCounter(
    bExecute := bCaseInvalid AND stMetsStatus.bNVDataInitOK,
    stCTDateTime := stMetsStatus.stCTDateTime,
    nCaseRejectID := stCaseQueue.stPrintCACData.CaseRejectID,
    aRejectCountersID := aRejectCountersID,
    aShiftRejectCounters := stShiftStatisticNV.aRejectCounters,
    aProdRejectCounters := stProdStatisticNV.aRejectCounters); // FB_KPI_CaseLevelCounter

// NETWORK 40
// Alarm for nConsecutiveRejects consecutive 1d scanner failures
fbRejectCount(
    CU := bCaseInvalid AND stMetsStatus.stPCMStatus.bEnableCaseLabels AND NOT (stMachineConfig.nConsecutiveCaseRejects = 0),
    RESET := NOT stMetsStatus.stPCMStatus.bEnableCaseLabels OR bCaseValid OR stMetsStatus.bShortReset OR stMachineConfig.nConsecutiveCaseRejects = 0,
    PV := stMachineConfig.nConsecutiveCaseRejects,
    CV => nRejectActualCount); // CTU
bAlarm_ConsecutiveCaseRejects S= fbRejectCount.Q AND NOT (stMachineConfig.nConsecutiveCaseRejects = 0);

// NETWORK 41
fbCaseValidationScanned(
    bInput := b01_ScanLabel AND NOT bCaseRejectedBeforeScanLabelSignal,
    bReset := stMetsStatus.stPCMStatus.bRSKUChanged OR stMetsStatus.stPCMStatus.bOpModeChanged OR stResetCaseInspectionHMI.bButtonState,
    nCounter := stCaseInspactionLogNV.nCaseValidationScanned); // FB_CTU32

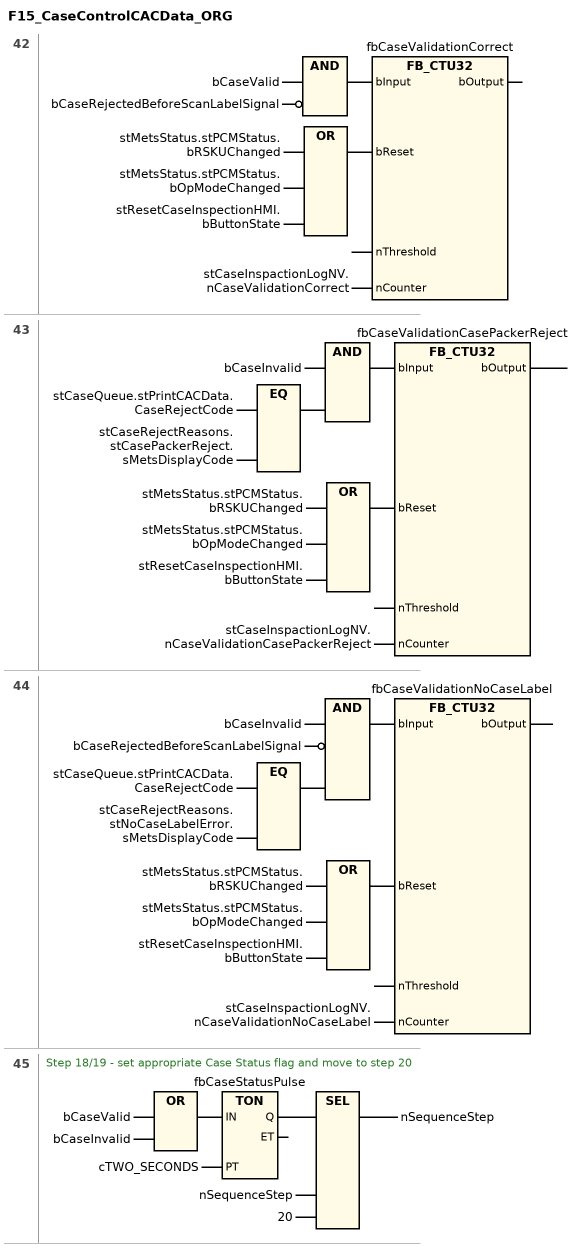
// NETWORK 42
fbCaseValidationCorrect(
    bInput := bCaseValid AND NOT bCaseRejectedBeforeScanLabelSignal,
    bReset := stMetsStatus.stPCMStatus.bRSKUChanged OR stMetsStatus.stPCMStatus.bOpModeChanged OR stResetCaseInspectionHMI.bButtonState,
    nCounter := stCaseInspactionLogNV.nCaseValidationCorrect); // FB_CTU32

// NETWORK 43
fbCaseValidationCasePackerReject(
    bInput := bCaseInvalid AND stCaseQueue.stPrintCACData.CaseRejectCode = stCaseRejectReasons.stCasePackerReject.sMetsDisplayCode,
    bReset := stMetsStatus.stPCMStatus.bRSKUChanged OR stMetsStatus.stPCMStatus.bOpModeChanged OR stResetCaseInspectionHMI.bButtonState,
    nCounter := stCaseInspactionLogNV.nCaseValidationCasePackerReject); // FB_CTU32

// NETWORK 44
fbCaseValidationNoCaseLabel(
    bInput := bCaseInvalid AND NOT bCaseRejectedBeforeScanLabelSignal AND stCaseQueue.stPrintCACData.CaseRejectCode = stCaseRejectReasons.stNoCaseLabelError.sMetsDisplayCode,
    bReset := stMetsStatus.stPCMStatus.bRSKUChanged OR stMetsStatus.stPCMStatus.bOpModeChanged OR stResetCaseInspectionHMI.bButtonState,
    nCounter := stCaseInspactionLogNV.nCaseValidationNoCaseLabel); // FB_CTU32

// NETWORK 45
// Step 18/19 - set appropriate Case Status flag and move to step 20
fbCaseStatusPulse(IN := bCaseValid OR bCaseInvalid, PT := cTWO_SECONDS); // TON
nSequenceStep := SEL(fbCaseStatusPulse.Q, nSequenceStep, 20);

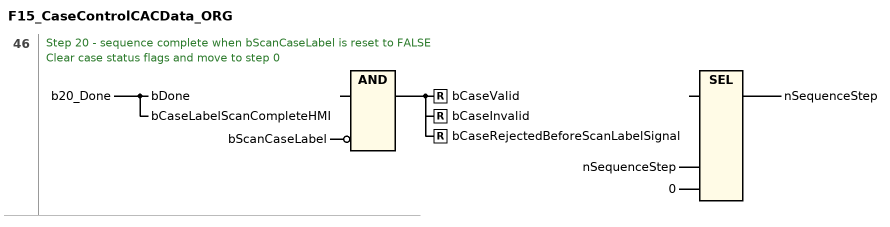
// NETWORK 46
// 					Step 20 - sequence complete when bScanCaseLabel is reset to FALSE
// Clear case status flags and move to step 0
//
bDone := b20_Done;
bCaseLabelScanCompleteHMI := b20_Done;
_w3 := b20_Done AND NOT bScanCaseLabel;
bCaseValid R= _w3;
bCaseInvalid R= _w3;
bCaseRejectedBeforeScanLabelSignal R= _w3;
nSequenceStep := SEL(_w3, nSequenceStep, 0);

ACTION CodesGetItem:
IF stMetsStatus.stPCMStatus.nOutersPerCase > 0 AND stMetsStatus.stPCMStatus.nPacksPerOuter > 0 THEN

	sCaseSerialCode := F_CODE_GetItem(stCaseQueue.stPrintCACData.Barcode, eCodeAIType.SerialCode, stMachineConfig.stCodeInfo_Case);
	sFirstOuterInCase := F_CODE_GetItem(stCaseQueue.stPrintCACData.Outer[1].Barcode, eCodeAIType.SerialCode, stMachineConfig.stCodeInfo_Outer);
	sLastOuterInCase := F_CODE_GetItem(stCaseQueue.stPrintCACData.Outer[stMetsStatus.stPCMStatus.nOutersPerCase].Barcode, eCodeAIType.SerialCode, stMachineConfig.stCodeInfo_Outer);
	sFirstPackSerialCode := F_CODE_GetItem(stCaseQueue.stPrintCACData.Outer[1].PackCode[1], eCodeAIType.SerialCode, stMachineConfig.stCodeInfo_Pack);
	sLastPackSerialCode := F_CODE_GetItem(stCaseQueue.stPrintCACData.Outer[stMetsStatus.stPCMStatus.nOutersPerCase].PackCode[stMetsStatus.stPCMStatus.nPacksPerOuter], eCodeAIType.SerialCode, stMachineConfig.stCodeInfo_Pack);

	sFirstOuterInCase	:= RIGHT(sFirstOuterInCase,7);
	sLastOuterInCase	:= RIGHT(sLastOuterInCase,7);
	sFirstPackSerialCode	:= RIGHT(sFirstPackSerialCode,7);
	sLastPackSerialCode	:= RIGHT(sLastPackSerialCode,7);

	sPrintCaseContent  := F_CONCAT9('Init OUT ID [',sFirstOuterInCase, '] ; Last OUT ID [', sLastOuterInCase,  '] ; Init PK ID [',sFirstPackSerialCode, '] ; Last PK ID [', sLastPackSerialCode,']');
END_IF
END_ACTION

END_PROGRAM

// ---- POUs/_Exclude/v2/FB_CAC_WriteToArchive_v2.TcPOU
(* reads CAC files from CAC folder, deletes OAC file and copies CAC file into Archive *)
FUNCTION_BLOCK FB_CAC_WriteToArchive_v2
VAR_INPUT
	bExecute				: BOOL;		(* set TRUE to archive OAC files *)
	sCaseFilename			: T_CAC_Filename;
	sLocalCACPath			: T_MaxString;	(* path to CaseTrace CAC folder *)
	sLocalOACPath			: T_MaxString;	(* path to CaseTrace OAC folder *)
	sLocalOCVPath			: T_MaxString;	(* path to CaseTrace OAC folder *)
	sSystemTime			: TIMESTRUCT;
	bUseInterimCodeForValidation	: BOOL;
END_VAR
VAR_IN_OUT
	stCodeInfo_Pack			: ST_CodeInfo;
	stCodeInfo_Intermediate	: ST_CodeInfo;
	stCodeInfo_Case			: ST_CodeInfo;
	stProductInstruction		: ST_PCM_Status;
	stPrintCACData			: ST_CAC_Data;
END_VAR
VAR_OUTPUT
	bDone 					: BOOL;		(* TRUE = OAC archive complete *)
	bBusy 					: BOOL;		(* TRUE = OAC archive active *)
	bError 					: BOOL;		(* TRUE = OAC archive error *)
	nErrorID				: UDINT;	(* error code *)
	stCACData				: ST_CAC_Data;
	nOACFilesDeleted		: UDINT;
	nOCVFilesDeleted		: UDINT;
	sCACFile				: T_CAC_Filename;
	bCACValid						: BOOL;
END_VAR
VAR
	fbExecute				: R_TRIG;
	eState					: E_CAC_State;
	eErrorState				: E_CAC_State;

	sDateFolder			: STRING(11);
	sTargetPath			: STRING(255);

	bWriteCACFileExec		: BOOL;
	fbWriteCACFile			: FB_CAC_WriteFile_v2;

	nOuterIndex			: INT;
	sOACFile				: T_OAC_Filename;
	sOCVFile				: T_OAC_Filename;
	aOCVFileCodeName	: ARRAY[1..2] OF T_MaxString;

	bDeleteFileExec		: BOOL;
	fbDeleteFile			: FB_FileDelete;
	sDeletePathName		: STRING(255);
	ftDeleteFileDone		: F_TRIG;

END_VAR

(* monitor bExecute for rising edge *)
fbExecute(CLK := bExecute);

CASE eState OF

	(* idle *)
	E_CAC_IDLE:

		(* rising edge of bExecute *)
		IF fbExecute.Q = TRUE THEN

			(* update outputs *)
			bDone := FALSE;
			bBusy := TRUE;
			bError := FALSE;
			nErrorID := 0;

			sDateFolder	:= '';
			sTargetPath 	:= '';
			bCACValid		:= FALSE;

			MEMSET(ADR(stCACData), 16#00, SIZEOF(stCACData));
			MEMMOVE(ADR(stCACData), ADR(stPrintCACData),  SIZEOF(stCACData));

			nOACFilesDeleted := 0;
			nOCVFilesDeleted := 0;

			eState := E_CAC_WRITEDATA;

		(* bExecute has been reset *)
		ELSIF bExecute = FALSE THEN

			(* clear outputs *)
			bDone := FALSE;
			bBusy := FALSE;
			bError := FALSE;
			nErrorID := 0;
		END_IF

(*****************************************************************************************)

	(* create folders *)
	E_CAC_WRITEDATA:

		(* Set up CAC target path to store file*)
		IF F_ToUCase(stCACData.CaseRejectCode) = 'OK' THEN


			IF stCodeInfo_Case.stProductionOrder.nListPosition = 0 THEN

				sDateFolder := stProductInstruction.sRetailSKU;

			ELSIF stProductInstruction.sProductionOrder  <> '' THEN

				sDateFolder := stProductInstruction.sProductionOrder;
			ELSE
				sDateFolder := F_SYSTEM_SystemTimeToFolderName(sSystemTime);
			END_IF

			sCACFile 		:= sCaseFilename;
			sTargetPath 	:= F_CONCAT4(sLocalCACPath, 'Archive\', sDateFolder, '\');
		ELSE

			sCACFile 		:= CONCAT('Err', sCaseFilename);
			sTargetPath	:= CONCAT(sLocalCACPath, 'Error\');
		END_IF

		bWriteCACFileExec				:= TRUE;
		(* Write CAC to archive folder *)
		(*fbWriteCACFile(
			bExecute					:= TRUE,
			bOverwrittenCAC			:= FALSE,
			sTargetPath				:= sTargetPath,
			sCACFile					:= sCACFile,
			tTimeout					:= cTHREE_SECONDS,
			stCACData					:= stCACData
			);*)

		IF fbWriteCACFile.bDone THEN

			bCACValid	:= fbWriteCACFile.bCACValid;

			IF NOT fbWriteCACFile.bError THEN

				IF stCACData.CodingAndTrackingMode >= 7 AND bCACValid THEN

						(* OAC file management required, generate OAC file name *)
						sOACFile := F_CONCAT3('OAC_', F_OUTER_BarcodeToHex(stCACData.Outer[1].Barcode), '.xml');

						nOuterIndex := 1;

						eState := E_CAC_DELETEOAC;

					(* OAC data was not active when CAC file was produced *)
					ELSE
	
						(* OAC file management not required*)
						eState := E_CAC_DONE;
					END_IF

			(* write CAC error *)
			ELSE

				(* update outputs *)
				bError := TRUE;
				nErrorID := fbWriteCACFile.nErrorID;
				eErrorState := eState;

				eState := E_CAC_DONE;
			END_IF

			bWriteCACFileExec				:= FALSE;
			(* close off fbCreateFolder *)
			(*fbWriteCACFile(
				bExecute 	:= FALSE,
				stCACData	:= stCACData
				);*)
		END_IF

	(* delete OAC files *)
	E_CAC_DELETEOAC:

		sDeletePathName 	:= CONCAT(sLocalOACPath, sOACFile);
		bDeleteFileExec	:= TRUE;
		(* delete OAC file *)
		(*fbDeleteFile(
			sNetId		:= '',
			sPathName	:= CONCAT(sLocalOACPath, sOACFile),
			ePath		:= PATH_GENERIC,
			bExecute	:= TRUE,
			tTimeout	:= cTHREE_SECONDS
			);*)

		(* delete file complete *)
		IF ftDeleteFileDone.Q THEN

			(* delete file completed OK *)
			IF NOT fbDeleteFile.bError  THEN

				(* update counter *)
				nOACFilesDeleted := nOACFilesDeleted + 1;
			ELSE

				(* update outputs *)
				bError := fbDeleteFile.bError;
				nErrorID := fbDeleteFile.nErrId;
				eErrorState := eState;
			END_IF

			 IF stProductInstruction.nOutersPerCase = stCACData.NumberOfOuters THEN
				(* all OAC files archived *)
				IF nOuterIndex = stCACData.NumberOfOuters THEN

					aOCVFileCodeName[1]	:=	F_CODE_GetItem(stCACData.Outer[1].AggregationCodes[1] , eCodeAIType.SerialCode,
																	SEL(bUseInterimCodeForValidation, stCodeInfo_Pack, stCodeInfo_Intermediate));
					sOCVFile := F_CONCAT3('OCV_', F_CodeToHex(aOCVFileCodeName[1]), '.xml');
					nOuterIndex := 1;
	
					eState := E_CAC_DELETEOCV1;

				ELSE
				(* more OAC files to be archived *)
					nOuterIndex := LIMIT(1, nOuterIndex + 1, stProductInstruction.nOutersPerCase);
					(* generate next OAC file name *)
					sOACFile := F_CONCAT3('OAC_', F_OUTER_BarcodeToHex(stCACData.Outer[nOuterIndex].Barcode), '.xml');
				END_IF
			ELSE
				eState := E_CAC_DONE;
			END_IF
			(* close off fbDeleteFile *)
			bDeleteFileExec	:= FALSE;
			(*fbDeleteFile(bExecute := FALSE);*)
		END_IF

	E_CAC_DELETEOCV1:
		(* delete 1st OCV file *)

		sDeletePathName := CONCAT(sLocalOCVPath, sOCVFile);
		bDeleteFileExec	:= TRUE;

		(*fbDeleteFile(
			sNetId		:= '',
			sPathName	:= CONCAT(sLocalOCVPath, sOCVFile),
			ePath		:= PATH_GENERIC,
			bExecute	:= TRUE,
			tTimeout	:= cTHREE_SECONDS
		);*)

		(* delete file complete *)
		IF ftDeleteFileDone.Q THEN

			(* delete file completed OK *)
			IF NOT fbDeleteFile.bError  THEN

				(* update counter *)
				nOCVFilesDeleted := nOCVFilesDeleted + 1;

			ELSE

				(* update outputs *)
				bError := fbDeleteFile.bError;
				nErrorID := fbDeleteFile.nErrId;
				eErrorState := eState;
			END_IF

			 IF stProductInstruction.nOutersPerCase = stCACData.NumberOfOuters THEN
			(* all OCV files archived *)
				IF nOuterIndex = stCACData.NumberOfOuters THEN

					aOCVFileCodeName[2]	:=	F_CODE_GetItem(stCACData.Outer[1].AggregationCodes[2] , eCodeAIType.SerialCode,   stCodeInfo_Pack); (*no reason to have 2 diffrent intermediate codes*)
					sOCVFile := F_CONCAT3('OCV_', F_CodeToHex(aOCVFileCodeName[2]), '.xml');
					nOuterIndex := 1;

					eState := SEL(bUseInterimCodeForValidation, E_CAC_DELETEOCV2, E_CAC_DONE);
	
				ELSE
				(* more OCV files to be archived *)
					nOuterIndex := LIMIT(1, nOuterIndex + 1, stProductInstruction.nOutersPerCase);
					(* generate next OCV file name *)
					aOCVFileCodeName[1]	:=	F_CODE_GetItem(stCACData.Outer[nOuterIndex].AggregationCodes[1] , eCodeAIType.SerialCode,
																						SEL(bUseInterimCodeForValidation, stCodeInfo_Pack, stCodeInfo_Intermediate));
					sOCVFile := F_CONCAT3('OCV_', F_CodeToHex(aOCVFileCodeName[1]), '.xml');
				END_IF
			ELSE
				eState := E_CAC_DONE;
			END_IF
			(* close off fbDeleteFile *)
			bDeleteFileExec	:= FALSE;
			(*fbDeleteFile(bExecute := FALSE);*)
		END_IF

	E_CAC_DELETEOCV2:
		(* delete 2nd OCV file *)
		sDeletePathName := CONCAT(sLocalOCVPath, sOCVFile);
		bDeleteFileExec	:= TRUE;

		(*fbDeleteFile(
			sNetId		:= '',
			sPathName	:= CONCAT(sLocalOCVPath, sOCVFile),
			ePath		:= PATH_GENERIC,
			bExecute	:= TRUE,
			tTimeout	:= cTHREE_SECONDS
			);*)

		(* delete file complete *)
		IF ftDeleteFileDone.Q THEN

			(* delete file completed OK *)
			IF NOT fbDeleteFile.bError  THEN

				(* update counter *)
				nOCVFilesDeleted := nOCVFilesDeleted + 1;
			ELSE

				(* update outputs *)
				bError := fbDeleteFile.bError;
				nErrorID := fbDeleteFile.nErrId;
				eErrorState := eState;
			END_IF

			IF stProductInstruction.nOutersPerCase = stCACData.NumberOfOuters THEN
				(* all OCV files archived *)
				IF nOuterIndex = stCACData.NumberOfOuters THEN
	
					eState := E_CAC_DONE;
				ELSE
				(* more OCV files to be archived *)
					nOuterIndex := LIMIT(1, nOuterIndex + 1, stProductInstruction.nOutersPerCase);
					(* generate next OCV file name *)
					aOCVFileCodeName[2]	:=	F_CODE_GetItem(stCACData.Outer[nOuterIndex].AggregationCodes[2] , eCodeAIType.SerialCode,   stCodeInfo_Pack);
					sOCVFile := F_CONCAT3('OCV_', F_CodeToHex(aOCVFileCodeName[2]), '.xml');
				END_IF
			ELSE
				eState := E_CAC_DONE;
			END_IF
			(* close off fbDeleteFile *)
			bDeleteFileExec	:= FALSE;
			(*fbDeleteFile(bExecute := FALSE);*)
		END_IF

	(* complete *)
	E_CAC_DONE:

		(* update outputs *)
		bBusy := FALSE;
		bDone := TRUE;

		eState := E_CAC_IDLE;

(* unknown state *)
ELSE

	eState := E_CAC_IDLE;
END_CASE

(*********************************************************************************************)

fbWriteCACFile(
			bExecute					:= bWriteCACFileExec,
			bOverwrittenCAC			:= FALSE,
			sTargetPath				:= sTargetPath,
			sCACFile					:= sCACFile,
			tTimeout					:= cTHREE_SECONDS,
			stCACData					:= stCACData
			);

		fbDeleteFile(
			sNetId		:= '',
			sPathName	:= sDeletePathName,
			ePath		:= PATH_GENERIC,
			bExecute	:= bDeleteFileExec,
			tTimeout	:= cTHREE_SECONDS
			);

		ftDeleteFileDone(CLK:= fbDeleteFile.bBusy);

END_FUNCTION_BLOCK

// ---- POUs/_Exclude/v2/FB_CAC_WriteFile_v2.TcPOU
FUNCTION_BLOCK FB_CAC_WriteFile_v2
VAR_INPUT
	bExecute						: BOOL;
	bOverwrittenCAC				: BOOL;
	sTargetPath					: T_MaxString;
	sCACFile						: T_CAC_Filename;	(* CAC file name generated from stCACData *)
	tTimeout						: TIME := cTHREE_SECONDS;
END_VAR
VAR_IN_OUT
	stCACData						: ST_CAC_Data;
END_VAR
VAR_OUTPUT
	bDone							: BOOL;
	bBusy							: BOOL;
	bError							: BOOL;
	nErrorID						: UDINT;
	bCACValid						: BOOL;
	sFirstOuter						: T_OUTER_Barcode;
	sLastOuter						: T_OUTER_Barcode;
	bBufferOverflow				: BOOL;
	nMaxBufferSize				: UDINT;
END_VAR
VAR
	fbExecute						: R_TRIG;
	eState							: E_CAC_State;
	eErrorState						: E_CAC_State;

	aCACImage				: ARRAY[0..cMAX_FILE_BUFFER] OF BYTE;
	sString						: STRING(255);
	nStringLen					: INT;
	nCACByte					: UINT;
	nOuterIndex				: INT;
	nMaxCACImageSize		: UINT;
	nControlSize				: UINT;



	fbCreateFolder					: FB_CreateDir;

	hFileHandle					: UINT;
	fbOpenFile						: FB_FileOpen;

	fbBuildOACData				: FB_OAC_BuildXMLData;
	fbPopulateMinimalOuterData	: FB_CAC_PopulateMinimalOuterData;

	fbWriteFile						: FB_FileWrite;
	fbCloseFile						: FB_FileClose;
END_VAR

fbExecute(CLK := bExecute);

nMaxBufferSize := MAX(nCACByte, nMaxBufferSize);

CASE eState OF

	(* idle *)
	E_CAC_IDLE:

		IF fbExecute.Q = TRUE THEN

			(* update outputs *)
			bDone := FALSE;
			bBusy := TRUE;
			bError := FALSE;
			nErrorID := 0;

			(* initialise CAC byte and output image *)
			nCACByte := 0;
			MEMSET(ADR(aCACImage), 16#00, SIZEOF(aCACImage));
			nControlSize := 0;
			nMaxCACImageSize := SIZEOF(aCACImage);


			(* build CAC template header fields *)
			(* XML header *)
			sString := cXML_HEADER;
			nStringLen := LEN(sString);
			MEMMOVE(ADR(aCACImage[nCACByte]), ADR(sString), nStringLen);
			nCACByte := nCACByte + nStringLen;

			(* <Comment> tag *)
			sString := '<!--File CAC builder. Version 2.2.000 Relase 01.08.2024 PTR -->$R$N';
			AppendImageData();


			(* <Case> tag *)
			sString := '<Case>$R$N';
			AppendImageData();

			(* <Barcode> field *)
			sString := F_CONCAT3('$T<Barcode><![CDATA[', stCACData.Barcode, ']]></Barcode>$R$N');
			AppendImageData();

			(* <ProductionDate> field *)
			sString := F_CONCAT3('$T<ProductionDate>', stCACData.ProductionDate, '</ProductionDate>$R$N');
			AppendImageData();

			(* <ProductionTime> field *)
			sString := F_CONCAT3('$T<ProductionTime>', stCACData.ProductionTime, '</ProductionTime>$R$N');
			AppendImageData();

			(* <ProductionTimeOffset> field *)
			sString := F_CONCAT3('$T<ProductionTimeOffset>', stCACData.ProductionTimeOffset, '</ProductionTimeOffset>$R$N');
			AppendImageData();

			(* <RetailSKU> field *)
			sString := F_CONCAT3('$T<RetailSKU>', stCACData.RetailSKU, '</RetailSKU>$R$N');
			AppendImageData();

			(* <CasePacker> tag *)
			sString := '$T<CasePacker>$R$N';
			AppendImageData();

			(* <ProductionSite> field *)
			sString := F_CONCAT3('$T$T<ProductionSite>', stCACData.CasePacker.ProductionSite, '</ProductionSite>$R$N');
			AppendImageData();

			(* <ProductionLine> field *)
			sString := F_CONCAT3('$T$T<ProductionLine>', stCACData.CasePacker.ProductionLine, '</ProductionLine>$R$N');
			AppendImageData();

			(* </CasePacker> tag *)
			sString := '$T</CasePacker>$R$N';
			AppendImageData();

			(* <CodingAndTrackingMode> field *)
			sString := F_CONCAT3('$T<CodingAndTrackingMode>', INT_TO_STRING(stCACData.CodingAndTrackingMode), '</CodingAndTrackingMode>$R$N');
			AppendImageData();

			(* <NumberOfOuters> field *)
			sString := F_CONCAT3('$T<NumberOfOuters>', INT_TO_STRING(stCACData.NumberOfOuters), '</NumberOfOuters>$R$N');
			AppendImageData();

			(* stCACData is valid *)
			IF F_ToUCase(stCACData.CaseRejectCode) = 'OK'  AND NOT bOverwrittenCAC THEN

				(* write valid CAC files to TEMP folder *)
				bCACValid := TRUE;

				(* first and last Outers in CAC file *)
				IF stCACData.NumberOfOuters <> 0 THEN
					sFirstOuter := stCACData.Outer[1].Barcode;
					sLastOuter := stCACData.Outer[stCACData.NumberOfOuters].Barcode;
				END_IF
				
			(* stCACData is invalid *)
			ELSE

				(* <CaseRejectCode> field *)
				sString := F_CONCAT3('$T<CaseRejectCode>', SEL(bOverwrittenCAC,  stCACData.CaseRejectCode, 'CACDataOver-written'), '</CaseRejectCode>$R$N');
				AppendImageData();

				(* <CaseRejectID> field *)
				sString := F_CONCAT3('$T<CaseRejectID>', UINT_TO_STRING(stCACData.CaseRejectID), '</CaseRejectID>$R$N');
				AppendImageData();

				(* generate CAC filename and target path for ErrCAC files *)
				bCACValid := FALSE;

				(* reset first and last Outers *)
				sFirstOuter := '';
				sLastOuter := '';
			END_IF

			(* first Outer to be added to aCACImage *)
			nOuterIndex := 1;

			eState := E_CAC_CREATEFOLDER;

		(* bExecute has been reset *)
		ELSIF bExecute = FALSE THEN

			(* update outputs *)
			bDone := FALSE;
			bBusy := FALSE;
			bError := FALSE;
			nErrorID := 0;
		END_IF

	E_CAC_CREATEFOLDER:

		(* create date archive folder *)
		fbCreateFolder(
			sNetId		:= '',
			sPathName	:= sTargetPath,
			ePath		:= PATH_GENERIC,
			bExecute	:= TRUE,
			tTimeout	:= T#1s
		);

		(* create folder complete *)
		IF fbCreateFolder.bBusy = FALSE THEN

			(* create folder completed OK or folder already exists *)
			IF fbCreateFolder.bError = FALSE OR (fbCreateFolder.bError = TRUE AND fbCreateFolder.nErrId = 16#70C) THEN

				eState := E_CAC_OPENFILE;

			(* create folder error *)
			ELSE

				(* update outputs *)
				bError := TRUE;
				nErrorID := fbCreateFolder.nErrId;
				eErrorState := eState;

				eState := E_CAC_DONE;
			END_IF

			(* close off fbCreateFolder *)
			fbCreateFolder(bExecute := FALSE);
		END_IF

	(* open CAC file for writing *)
	E_CAC_OPENFILE:

		fbOpenFile(
			sNetId		:= '',
			sPathName	:= CONCAT(sTargetPath, sCACFile),
			nMode		:= FOPEN_MODEWRITE OR FOPEN_MODEBINARY,
			ePath		:= PATH_GENERIC,
			bExecute	:= TRUE,
			tTimeout	:= T#1s
		);

		(* open file complete *)
		IF fbOpenFile.bBusy = FALSE THEN

			(* open file completed OK *)
			(*	OACdata now required in all modes	*)
			IF fbOpenFile.bError = FALSE THEN

				(* file handle *)
				hFileHandle := fbOpenFile.hFile;

				(* OAC data required in CAC file *)
				IF stCACData.CodingAndTrackingMode >= 7 THEN

					eState := E_CAC_BUILDXMLIMAGE;

				(* OAC data not required in CAC file *)
				ELSE
					(* Fill in  Minimal data into stCACData.Outer*)
					fbPopulateMinimalOuterData(
					bExecute := TRUE,
					nNumberofOuters := stCACData.NumberOfOuters,
					stCACData := stCACData
					);

					IF fbPopulateMinimalOuterData.bDone THEN
						eState := E_CAC_BUILDXMLIMAGE;
					END_IF
				END_IF

			(* open file error *)
			ELSE

				bError := TRUE;
				nErrorID := fbOpenFile.nErrID;
				eErrorState := eState;

				eState := E_CAC_DONE;
			END_IF

			(* close off fbOpenFile *)
			fbOpenFile(bExecute := FALSE);
		END_IF


	(* build XML image for CAC data *)
	E_CAC_BUILDXMLIMAGE:

	(* Reset *)
		fbPopulateMinimalOuterData(
			bExecute := FALSE,
			nNumberofOuters := stCACData.NumberOfOuters,
			stCACData := stCACData
		);

		(* build template for Outer *)
		fbBuildOACData(
			bExecute		:= TRUE,
			bAddXMLHEader	:= FALSE,
			nTabIndent		:= 1,
			nOuterIndex		:= nOuterIndex,
			stOACData		:= stCACData.Outer[nOuterIndex]
		);

		(* build OAC data complete *)
		IF fbBuildOACData.bDone = TRUE THEN

			(* aCACImage has room for OAC data and trailing </Case> tag (if required) *)
			IF SIZEOF(aCACImage) - nCACByte - LEN('</Case>') > fbBuildOACData.nOACByte THEN

				nControlSize := nControlSize + fbBuildOACData.nOACByte;
				IF nControlSize <  nMaxCACImageSize AND stCACData.NumberOfOuters <> 0 THEN
					MEMMOVE(ADR(aCACImage[nCACByte]), ADR(fbBuildOACData.arrOACImage), fbBuildOACData.nOACByte);
					nCACByte := nCACByte + fbBuildOACData.nOACByte;
				ELSE
					bBufferOverflow	:=TRUE;
					eState := E_CAC_CLOSEFILE;
					(*bDone := TRUE;*)
					(*RETURN;*)
				END_IF

				(* last Outer in Case *)
				IF nOuterIndex = stCACData.NumberOfOuters OR  stCACData.NumberOfOuters = 0THEN

					(* append </Case> tag *)
					sString := '</Case>';
					AppendImageData();
				END_IF
			END_IF

			eState := E_CAC_WRITEXMLIMAGE;

			(* close off fbBuildOACData *)
			fbBuildOACData(bExecute := FALSE);
		END_IF

	(* write CAC file template *)
	E_CAC_WRITEXMLIMAGE:

		(* write data to file *)
		fbWriteFile(
			sNetId		:= '',
			hFile		:= hFileHandle,
			pWriteBuff	:= ADR(aCACImage),
			cbWriteLen	:= nCACByte,
			bExecute	:= TRUE,
			tTimeout	:= tTimeout
		);

		(* write file complete *)
		IF fbWriteFile.bBusy = FALSE THEN

			(* write file completed OK *)
			IF fbWriteFile.bError = FALSE THEN

				(* OAC required and more OAC data to be written *)
				IF nOuterIndex < stCACData.NumberOfOuters THEN

					(* re-initialise CAC byte and output image *)
					nCACByte := 0;
					nControlSize := 0;
					MEMSET(ADR(aCACImage), 16#00, SIZEOF(aCACImage));
					(* next Outer in Case *)
					nOuterIndex := nOuterIndex + 1;

					eState := E_CAC_BUILDXMLIMAGE;

				(* all Outers added to CAC file or Outer data not required *)
				ELSE
					eState := E_CAC_CLOSEFILE;
				END_IF
			(* write file error *)
			ELSE

				bError := TRUE;
				nErrorID := fbWriteFile.nErrID;
				eErrorState := eState;

				eState := E_CAC_CLOSEFILE;
			END_IF

			(* close off fbWriteFile *)
			fbWriteFile(bExecute := FALSE);
		END_IF


	(* close CAC template *)
	E_CAC_CLOSEFILE:

		(* close file *)
		fbCloseFile(
			sNetId		:= '',
			hFile		:= hFileHandle,
			bExecute	:= TRUE,
			tTimeout	:= T#1s
		);

		(* close file complete *)
		IF fbCloseFile.bBusy = FALSE THEN

			(* close file completed OK and no file write error *)
			IF fbCloseFile.bError = FALSE AND bError = FALSE THEN

				eState := E_CAC_DONE;

			(* close file error or previous error with file write *)
			ELSE

				(* no previous error *)
				IF bError = FALSE THEN

					(* update error status *)
					bError := FALSE;
					nErrorID := fbCloseFile.nErrId;
					eErrorState := eState;
				END_IF

				eState := E_CAC_DONE;
			END_IF

			(* close off fbCloseFile *)
			fbCloseFile(bExecute := FALSE);
		END_IF

	(* complete *)
	E_CAC_DONE:

		bDone := TRUE;
		bBusy := FALSE;

		eState := E_CAC_IDLE;

(* unknown state *)
ELSE

	eState := E_CAC_IDLE;
END_CASE

ACTION AppendImageData:
nStringLen := LEN(sString);
nControlSize := nControlSize + nStringLen;
IF nControlSize <  nMaxCACImageSize THEN
	MEMMOVE(ADR(aCACImage[nCACByte]), ADR(sString), nStringLen);
	nCACByte := nCACByte + nStringLen;
ELSE
	bBufferOverflow	:=TRUE;
	bDone := TRUE;
	(*RETURN;*)
END_IF
END_ACTION

END_FUNCTION_BLOCK

// ---- POUs/_Exclude/v1/FB_CAC_PopulateMinimalOuterData.TcPOU
FUNCTION_BLOCK FB_CAC_PopulateMinimalOuterData
VAR_INPUT
	bExecute						: BOOL;
	nNumberofOuters					: INT;
END_VAR
VAR_IN_OUT
	stCACData						: ST_CAC_Data;
END_VAR
VAR_OUTPUT
	bDone: BOOL;
	bBusy: BOOL;
	bError: BOOL;
END_VAR
VAR
	fbExecute: R_TRIG;
	iOuter: INT;
END_VAR

fbExecute(CLK := bExecute);


IF fbExecute.Q = TRUE THEN

			(* update outputs *)
			bDone := FALSE;
			bBusy := TRUE;
			bError := FALSE;
END_IF

IF bBusy THEN

	FOR iOuter := 1TO nNumberofOuters DO
		stCACData.Outer[iOuter].CodingAndTrackingMode := 0;
		stCACData.Outer[iOuter].NumberOfPacks := 0;
		stCACData.Outer[iOuter].AcceptanceLevel := 0;
		stCACData.Outer[iOuter].NumberOfLinkedPacks := 0;
	END_FOR

	bDone := TRUE;

END_IF

IF bDone THEN
	bBusy := FALSE;
END_IF

END_FUNCTION_BLOCK

// ---- POUs/_Exclude/F21_ContentHandScanner_ORG.TcPOU
PROGRAM F21_ContentHandScanner_ORG
VAR
	fbBarcodeType			: FB_SYSTEM_BarcodeType;

	bPackBarcode					: BOOL;
	bOuterIntermediateBarcode		: BOOL;
	bOuterBarcode					: BOOL;
	bCaseBarcode					: BOOL;
	sPackBarcode					: T_PACK_Barcode;
	sOuterIntermediateBarcode		:  T_MaxString;
	sOuterBarcode					: T_OUTER_Barcode;
	sCaseBarcode					: T_CASE_Barcode;

	fbSearchCaseContent	: FB_SYSTEM_SearchBarcode;

	fbFindOACFile			: FB_OAC_FindFile;
	fbFindOCVFile			: FB_OCV_FindFile;
	stOACData				: ST_OAC_Data;
	strCode				: T_PACK_Barcode;
	strOACFile				: T_OAC_Filename;
	strOCVFile				: T_OCV_Filename;


	fbMoveCACFromArchive	: FB_CAC_MoveFromArchive;

	strCACFile				: T_CAC_Filename;

	bOACFound: BOOL;
	bOCVFound: BOOL;
	bOCVValid: BOOL;
	strOuterCodeAI:			STRING(255);
	(*strPackCodeAI:			STRING(255);*)

	bValidateForOCVDataExistDone :BOOL;
	bValidateForRefeedDone: BOOL;
	bValidateForRefeedOK: BOOL;

	rtrigValidateOCVForDataExistValid			: R_TRIG;
	rtrigValidateOCVForDataExistInvalid			: R_TRIG;
	rtrigValidateOCVForDataNotExist			: R_TRIG;
	tofValidateOCVForDataExisValid			: TOF;
	tofValidateOCVForDataExisInvalid			: TOF;
	tofValidateOCVForDataNotExis				: TOF;


	rtrigValidateOACForRefeedDoneValid		: R_TRIG;
	rtrigValidateOACForRefeedDoneInvalid		: R_TRIG;
	rtrigValidateOACForDataNotExist			: R_TRIG;
	tofValidateOACForRefeedValid			: TOF;
	tofValidateOACForRefeedInvalid			: TOF;
	tofValidateOACForDataNotExis				: TOF;

	rtrigRestoreCACFileDoneValid: R_TRIG;
	rtrigRestoreCACFileDoneInvalid: R_TRIG;
	tofRestoreCACFileValid: TOF;
	tofRestoreCACFileInvalid: TOF;

END_VAR

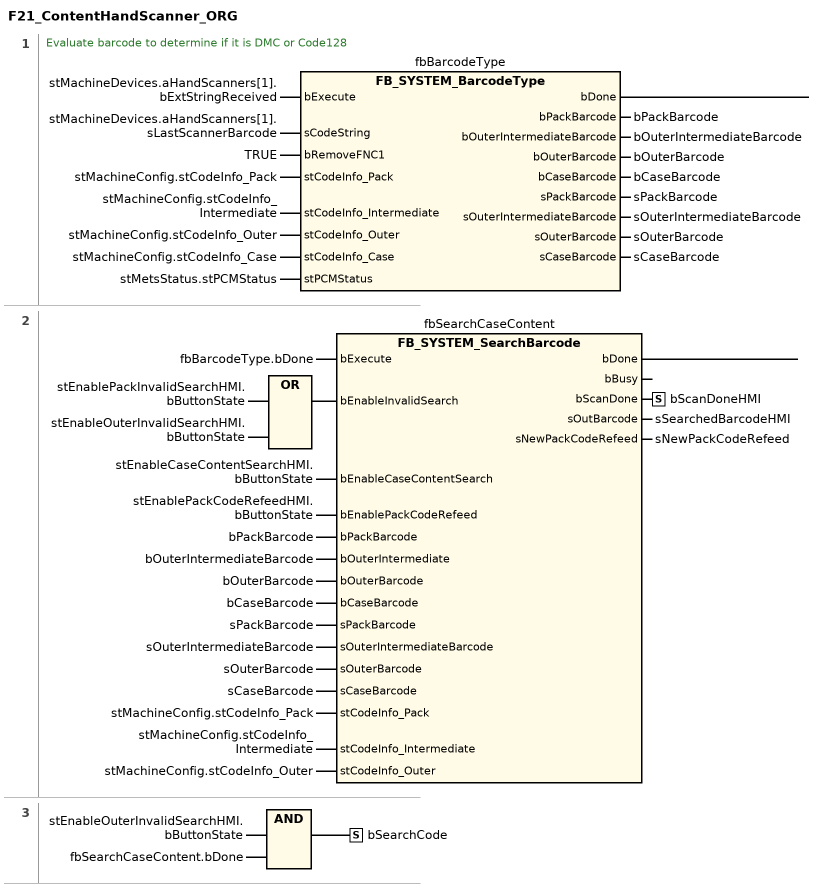
// NETWORK 1
// Evaluate barcode to determine if it is DMC or Code128
fbBarcodeType(
    bExecute := stMachineDevices.aHandScanners[1].bExtStringReceived,
    sCodeString := stMachineDevices.aHandScanners[1].sLastScannerBarcode,
    bRemoveFNC1 := TRUE,
    stCodeInfo_Pack := stMachineConfig.stCodeInfo_Pack,
    stCodeInfo_Intermediate := stMachineConfig.stCodeInfo_Intermediate,
    stCodeInfo_Outer := stMachineConfig.stCodeInfo_Outer,
    stCodeInfo_Case := stMachineConfig.stCodeInfo_Case,
    stPCMStatus := stMetsStatus.stPCMStatus,
    bPackBarcode => bPackBarcode,
    bOuterIntermediateBarcode => bOuterIntermediateBarcode,
    bOuterBarcode => bOuterBarcode,
    bCaseBarcode => bCaseBarcode,
    sPackBarcode => sPackBarcode,
    sOuterIntermediateBarcode => sOuterIntermediateBarcode,
    sOuterBarcode => sOuterBarcode,
    sCaseBarcode => sCaseBarcode); // FB_SYSTEM_BarcodeType

// NETWORK 2
fbSearchCaseContent(
    bExecute := fbBarcodeType.bDone,
    bEnableInvalidSearch := stEnablePackInvalidSearchHMI.bButtonState OR stEnableOuterInvalidSearchHMI.bButtonState,
    bEnableCaseContentSearch := stEnableCaseContentSearchHMI.bButtonState,
    bEnablePackCodeRefeed := stEnablePackCodeRefeedHMI.bButtonState,
    bPackBarcode := bPackBarcode,
    bOuterIntermediate := bOuterIntermediateBarcode,
    bOuterBarcode := bOuterBarcode,
    bCaseBarcode := bCaseBarcode,
    sPackBarcode := sPackBarcode,
    sOuterIntermediateBarcode := sOuterIntermediateBarcode,
    sOuterBarcode := sOuterBarcode,
    sCaseBarcode := sCaseBarcode,
    stCodeInfo_Pack := stMachineConfig.stCodeInfo_Pack,
    stCodeInfo_Intermediate := stMachineConfig.stCodeInfo_Intermediate,
    stCodeInfo_Outer := stMachineConfig.stCodeInfo_Outer,
    sOutBarcode => sSearchedBarcodeHMI,
    sNewPackCodeRefeed => sNewPackCodeRefeed); // FB_SYSTEM_SearchBarcode
bScanDoneHMI S= fbSearchCaseContent.bScanDone;

// NETWORK 3
bSearchCode S= stEnableOuterInvalidSearchHMI.bButtonState AND fbSearchCaseContent.bDone;

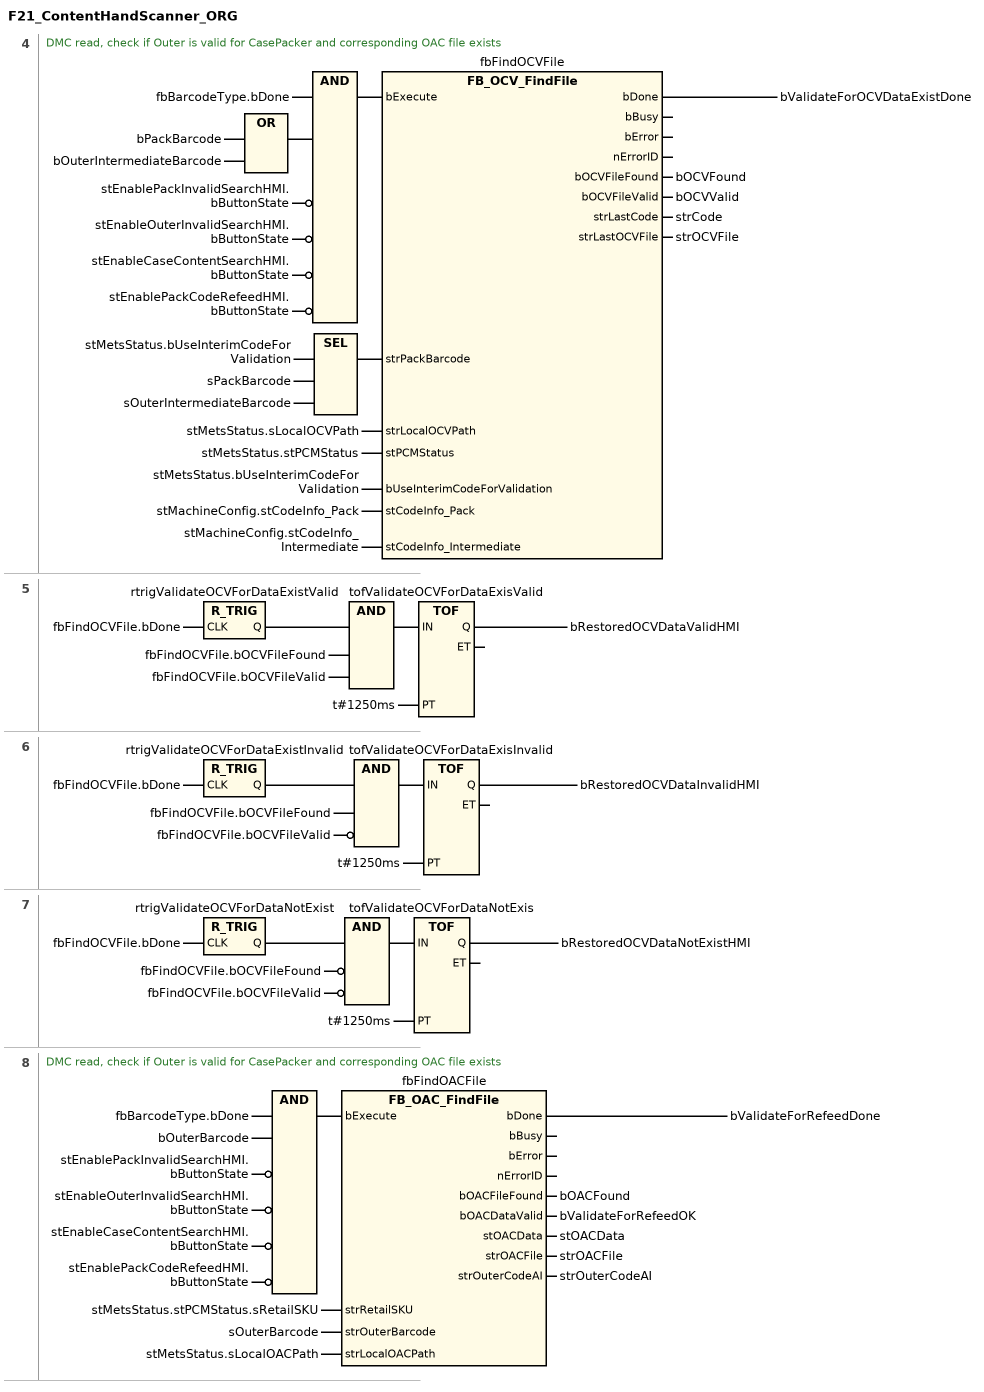
// NETWORK 4
// DMC read, check if Outer is valid for CasePacker and corresponding OAC file exists
fbFindOCVFile(
    bExecute := fbBarcodeType.bDone AND (bPackBarcode OR bOuterIntermediateBarcode) AND NOT stEnablePackInvalidSearchHMI.bButtonState AND NOT stEnableOuterInvalidSearchHMI.bButtonState AND NOT stEnableCaseContentSearchHMI.bButtonState AND NOT stEnablePackCodeRefeedHMI.bButtonState,
    strPackBarcode := SEL(stMetsStatus.bUseInterimCodeForValidation, sPackBarcode, sOuterIntermediateBarcode),
    strLocalOCVPath := stMetsStatus.sLocalOCVPath,
    stPCMStatus := stMetsStatus.stPCMStatus,
    bUseInterimCodeForValidation := stMetsStatus.bUseInterimCodeForValidation,
    stCodeInfo_Pack := stMachineConfig.stCodeInfo_Pack,
    stCodeInfo_Intermediate := stMachineConfig.stCodeInfo_Intermediate,
    bOCVFileFound => bOCVFound,
    bOCVFileValid => bOCVValid,
    strLastCode => strCode,
    strLastOCVFile => strOCVFile); // FB_OCV_FindFile
bValidateForOCVDataExistDone := fbFindOCVFile.bDone;

// NETWORK 5
rtrigValidateOCVForDataExistValid(CLK := fbFindOCVFile.bDone); // R_TRIG
tofValidateOCVForDataExisValid(IN := rtrigValidateOCVForDataExistValid.Q AND fbFindOCVFile.bOCVFileFound AND fbFindOCVFile.bOCVFileValid, PT := t#1250ms); // TOF
bRestoredOCVDataValidHMI := tofValidateOCVForDataExisValid.Q;

// NETWORK 6
rtrigValidateOCVForDataExistInvalid(CLK := fbFindOCVFile.bDone); // R_TRIG
tofValidateOCVForDataExisInvalid(IN := rtrigValidateOCVForDataExistInvalid.Q AND fbFindOCVFile.bOCVFileFound AND NOT fbFindOCVFile.bOCVFileValid, PT := t#1250ms); // TOF
bRestoredOCVDataInvalidHMI := tofValidateOCVForDataExisInvalid.Q;

// NETWORK 7
rtrigValidateOCVForDataNotExist(CLK := fbFindOCVFile.bDone); // R_TRIG
tofValidateOCVForDataNotExis(IN := rtrigValidateOCVForDataNotExist.Q AND NOT fbFindOCVFile.bOCVFileFound AND NOT fbFindOCVFile.bOCVFileValid, PT := t#1250ms); // TOF
bRestoredOCVDataNotExistHMI := tofValidateOCVForDataNotExis.Q;

// NETWORK 8
// DMC read, check if Outer is valid for CasePacker and corresponding OAC file exists
fbFindOACFile(
    bExecute := fbBarcodeType.bDone AND bOuterBarcode AND NOT stEnablePackInvalidSearchHMI.bButtonState AND NOT stEnableOuterInvalidSearchHMI.bButtonState AND NOT stEnableCaseContentSearchHMI.bButtonState AND NOT stEnablePackCodeRefeedHMI.bButtonState,
    strRetailSKU := stMetsStatus.stPCMStatus.sRetailSKU,
    strOuterBarcode := sOuterBarcode,
    strLocalOACPath := stMetsStatus.sLocalOACPath,
    bOACFileFound => bOACFound,
    bOACDataValid => bValidateForRefeedOK,
    stOACData => stOACData,
    strOACFile => strOACFile,
    strOuterCodeAI => strOuterCodeAI); // FB_OAC_FindFile
bValidateForRefeedDone := fbFindOACFile.bDone;

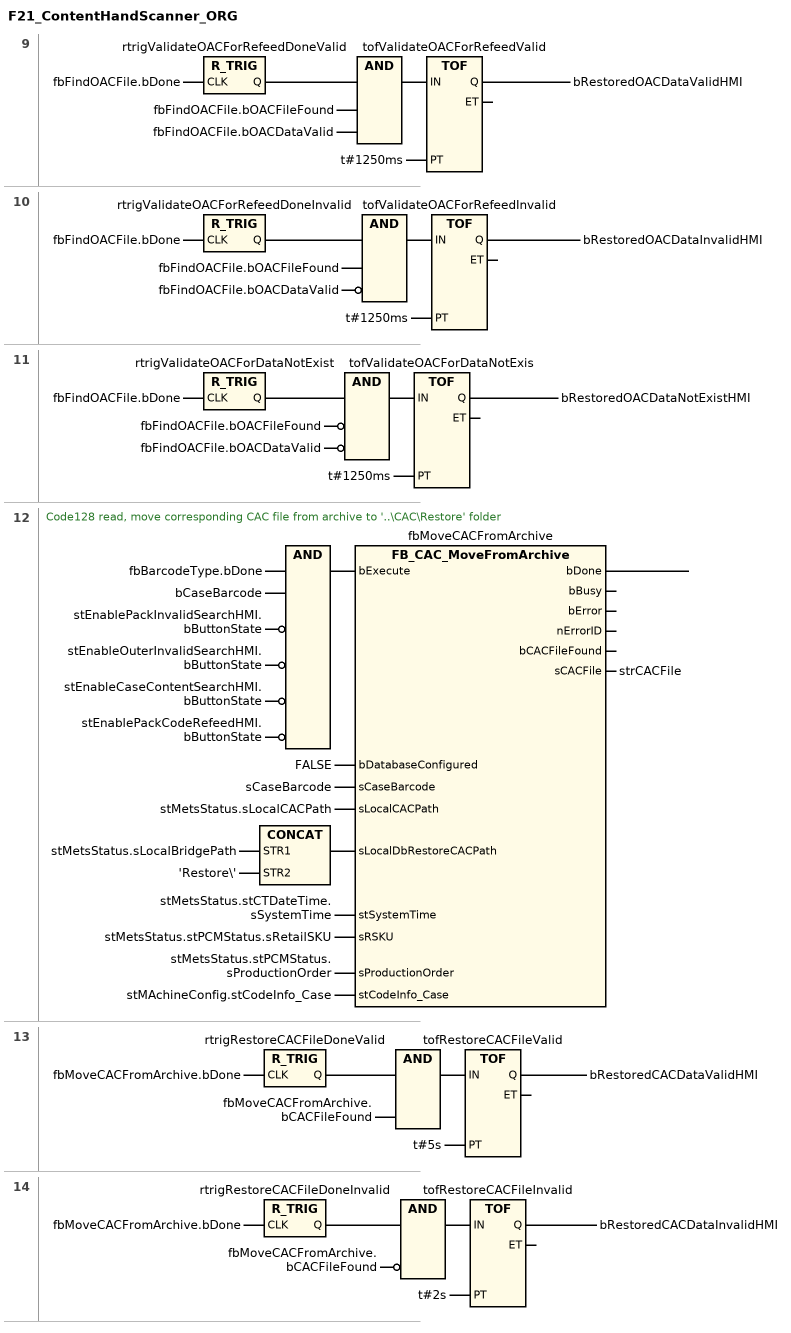
// NETWORK 9
rtrigValidateOACForRefeedDoneValid(CLK := fbFindOACFile.bDone); // R_TRIG
tofValidateOACForRefeedValid(IN := rtrigValidateOACForRefeedDoneValid.Q AND fbFindOACFile.bOACFileFound AND fbFindOACFile.bOACDataValid, PT := t#1250ms); // TOF
bRestoredOACDataValidHMI := tofValidateOACForRefeedValid.Q;

// NETWORK 10
rtrigValidateOACForRefeedDoneInvalid(CLK := fbFindOACFile.bDone); // R_TRIG
tofValidateOACForRefeedInvalid(IN := rtrigValidateOACForRefeedDoneInvalid.Q AND fbFindOACFile.bOACFileFound AND NOT fbFindOACFile.bOACDataValid, PT := t#1250ms); // TOF
bRestoredOACDataInvalidHMI := tofValidateOACForRefeedInvalid.Q;

// NETWORK 11
rtrigValidateOACForDataNotExist(CLK := fbFindOACFile.bDone); // R_TRIG
tofValidateOACForDataNotExis(IN := rtrigValidateOACForDataNotExist.Q AND NOT fbFindOACFile.bOACFileFound AND NOT fbFindOACFile.bOACDataValid, PT := t#1250ms); // TOF
bRestoredOACDataNotExistHMI := tofValidateOACForDataNotExis.Q;

// NETWORK 12
// Code128 read, move corresponding CAC file from archive to '..\CAC\Restore' folder
fbMoveCACFromArchive(
    bExecute := fbBarcodeType.bDone AND bCaseBarcode AND NOT stEnablePackInvalidSearchHMI.bButtonState AND NOT stEnableOuterInvalidSearchHMI.bButtonState AND NOT stEnableCaseContentSearchHMI.bButtonState AND NOT stEnablePackCodeRefeedHMI.bButtonState,
    bDatabaseConfigured := FALSE,
    sCaseBarcode := sCaseBarcode,
    sLocalCACPath := stMetsStatus.sLocalCACPath,
    sLocalDbRestoreCACPath := CONCAT(STR1 := stMetsStatus.sLocalBridgePath, STR2 := 'Restore\'),
    stSystemTime := stMetsStatus.stCTDateTime.sSystemTime,
    sRSKU := stMetsStatus.stPCMStatus.sRetailSKU,
    sProductionOrder := stMetsStatus.stPCMStatus.sProductionOrder,
    stCodeInfo_Case := stMAchineConfig.stCodeInfo_Case,
    sCACFile => strCACFile); // FB_CAC_MoveFromArchive

// NETWORK 13
rtrigRestoreCACFileDoneValid(CLK := fbMoveCACFromArchive.bDone); // R_TRIG
tofRestoreCACFileValid(IN := rtrigRestoreCACFileDoneValid.Q AND fbMoveCACFromArchive.bCACFileFound, PT := t#5s); // TOF
bRestoredCACDataValidHMI := tofRestoreCACFileValid.Q;

// NETWORK 14
rtrigRestoreCACFileDoneInvalid(CLK := fbMoveCACFromArchive.bDone); // R_TRIG
tofRestoreCACFileInvalid(IN := rtrigRestoreCACFileDoneInvalid.Q AND NOT fbMoveCACFromArchive.bCACFileFound, PT := t#2s); // TOF
bRestoredCACDataInvalidHMI := tofRestoreCACFileInvalid.Q;

END_PROGRAM

// ---- POUs/_Exclude/OAC FBs/FB_OAC_FindFile.TcPOU
(* converts strOuterBarcode to OAC filename and loads data *)
FUNCTION_BLOCK FB_OAC_FindFile
VAR_INPUT
	bExecute				: BOOL;		(* set TRUE to load OAC file *)
	strRetailSKU 			: T_CodeRSKU;
	strOuterBarcode		: T_MaxString;	(* Outer barcode *)
	strLocalOACPath		: T_FolderPath;	(* local OAC path *)
END_VAR
VAR_OUTPUT
	bDone				: BOOL;		(* TRUE = find file complete *)
	bBusy				: BOOL;		(* TRUE = find file in progress *)
	bError				: BOOL;		(* TRUE = error occurred *)
	nErrorID			: UDINT;	(* error code *)
	bOACFileFound		: BOOL;		(* TRUE = OAC file found *)
	bOACDataValid			: BOOL;
	stOACData			: ST_OAC_Data;	(* OAC data for strOuterBarcode *)
	strOACFile			: T_OAC_Filename;	(* OAC filename *)
	strOuterCodeAI		:T_MaxString;
END_VAR
VAR
	fbExecute			: R_TRIG;
	eState				: E_OAC_State;
	fbReadFile			: FB_XmlSrvRead;
	fbDecodeGS1				: FB_SCANNER_DecodeGS1;
END_VAR

fbExecute(CLK := bExecute);


CASE eState OF

	(* idle *)
	E_OAC_IDLE:

		(* rising edge of bExecute *)
		IF fbExecute.Q = TRUE THEN

			(* initialise outputs *)
			bDone := FALSE;
			bBusy := TRUE;
			bError := FALSE;
			nErrorID := 0;
			strOACFile := '';
			(* convert strOuterBarcode to OAC filename *)
			bOACFileFound := FALSE;
			bOACDataValid	:= FALSE;
			MEMSET(ADR(stOACData), 16#00, SIZEOF(stOACData));

			(* generate OAC file name and clear data for last OAC file *)
				(*fbDecodeGS1(strGS1String := CONCAT(']d2',strOuterBarcode), bDontParseAsGS1 := FALSE, strBarcode => strOuterCodeAI);*)
			strOACFile := F_CONCAT3('OAC_', F_OUTER_BarcodeToHex(strOuterBarcode), '.xml');


			eState := E_OAC_READFILE;

		(* bExecute has been reset *)
		ELSIF bExecute = FALSE THEN

			(* reset outputs *)
			bDone := FALSE;
			bBusy := FALSE;
			bError := FALSE;
			nErrorID := 0;
		END_IF


	(* read OAC file *)
	E_OAC_READFILE:

		(* read OAC file *)
		fbReadFile(
			sNetId		:= '',
			ePath		:= PATH_GENERIC,
			nMode		:= XMLSRV_SKIPMISSING,
			pSymAddr	:= ADR(stOACData),
			cbSymSize	:= SIZEOF(stOACData),
			sFilePath	:= CONCAT(strLocalOACPath, strOACFile),
			sXPath		:= '/Outer',
			bExecute	:= TRUE,
			tTimeout	:= T#1s
		);

		(* read file complete *)
		IF fbReadFile.bBusy = FALSE THEN

			(* read file completed OK *)
			IF fbReadFile.bError = FALSE THEN

				(* OAC file exists *)
				bOACFileFound := TRUE;

					IF strRetailSKU = stOACData.RetailSKU  AND stOACData.OuterRejectCode = 'OK'    THEN
						(* OAC data is valid *)
						bOACDataValid := TRUE;
					END_IF

			(* read file failed *)
			ELSE

				(* update outputs *)
				bError := TRUE;
				nErrorID := fbReadFile.nErrId;
			END_IF

			eState := E_OAC_DONE;

			(* close off fbReadFile *)
			fbReadFile(bExecute := FALSE);
		END_IF


	(* complete *)
	E_OAC_DONE:

		(* update outputs *)
		bDone := TRUE;
		bBusy := FALSE;

		eState := E_OAC_IDLE;


(* unknown state *)
ELSE

	eState := E_OAC_IDLE;

	(* clear outputs *)
	bDone := FALSE;
	bBusy := FALSE;
	bError := FALSE;
	nErrorID := 0;
	strOACFile := '';
END_CASE

END_FUNCTION_BLOCK

// ---- POUs/_Exclude/OCV FBs/FB_OCV_FindFile.TcPOU
(* converts strOuterBarcode to OCV filename and loads data *)
FUNCTION_BLOCK FB_OCV_FindFile
VAR_INPUT
	bExecute				: BOOL;		(* set TRUE to load OCV file *)
	strPackBarcode			: T_PACK_Barcode;	(* Outer barcode *)
	strLocalOCVPath		: STRING(50);	(* local OCV path *)
	stPCMStatus			: ST_PCM_Status;
	bUseInterimCodeForValidation	: BOOL;
END_VAR
VAR_IN_OUT
	stCodeInfo_Pack			: ST_CodeInfo;
	stCodeInfo_Intermediate		: ST_CodeInfo;
END_VAR
VAR_OUTPUT
	bDone				: BOOL;		(* TRUE = find file complete *)
	bBusy				: BOOL;		(* TRUE = find file in progress *)
	bError				: BOOL;		(* TRUE = error occurred *)
	nErrorID				: UDINT;		(* error code *)
	bOCVFileFound		: BOOL;		(* TRUE = OCV file found *)
	bOCVFileValid		: BOOL;		(* TRUE - OCV file valide*)
	strLastCode			: T_PACK_Barcode;
	strLastOCVFile			: T_OCV_Filename;	(* OCV filename *)
END_VAR
VAR
	fbExecute				: R_TRIG;
	eState				: E_OCV_State;
	eCodeAIType			: E_CodeAIType;
	fbReadFile			: FB_XmlSrvRead;
	sOCVFound			: ST_OUTER_Status;
END_VAR

fbExecute(CLK := bExecute);

CASE eState OF

	(* idle *)
	E_OCV_IDLE:

		(* rising edge of bExecute *)
		IF fbExecute.Q = TRUE THEN

			(* initialise outputs *)
			bDone := FALSE;
			bBusy := TRUE;
			bError := FALSE;
			nErrorID := 0;

			(* convert strOuterBarcode to OAC filename *)
			bOCVFileFound := FALSE;
			bOCVFileValid := FALSE;
			MEMSET(ADR(strLastCode), 16#00, SIZEOF(strLastCode));
			strLastCode := strPackBarcode;

			strLastOCVFile := F_CONCAT3('OCV_', F_CodeToHex(F_CODE_GetItem(strPackBarcode , eCodeAIType.SerialCode,
																SEL(bUseInterimCodeForValidation, stCodeInfo_Pack, stCodeInfo_Intermediate))), '.xml');

			eState := E_OCV_READFILE;

		(* bExecute has been reset *)
		ELSIF bExecute = FALSE THEN

			(* reset outputs *)
			bDone := FALSE;
			bBusy := FALSE;
			bError := FALSE;
			nErrorID := 0;

			(*bOCVFileFound := FALSE;*)
			(*bOCVFileValide := FALSE;*)
		END_IF


	(* read OCV file *)
	E_OCV_READFILE:

		(* read OCV file *)
		fbReadFile(
			sNetId		:= '',
			ePath		:= PATH_GENERIC,
			nMode		:= XMLSRV_SKIPMISSING,
			pSymAddr	:= ADR(sOCVFound),
			cbSymSize	:= SIZEOF(sOCVFound),
			sFilePath		:= CONCAT(strLocalOCVPath, strLastOCVFile),
			sXPath		:= '/OCVPack',
			bExecute		:= TRUE,
			tTimeout		:= T#1s
		);

		(* read file complete *)
		IF fbReadFile.bBusy = FALSE THEN

			(* read file completed OK *)
			IF fbReadFile.bError = FALSE THEN

				(* OCV file exists *)
				bOCVFileFound := TRUE;

				IF sOCVFound.stOACData.NumberOfLinkedPacks >= stPCMStatus.nAcceptanceLevel THEN
					bOCVFileValid := TRUE;
				END_IF

			(* read file failed *)
			ELSE

				(* update outputs *)
				bError := TRUE;
				nErrorID := fbReadFile.nErrId;

			END_IF

			eState := E_OCV_DONE;

			(* close off fbReadFile *)
			fbReadFile(bExecute := FALSE);
		END_IF


	(* complete *)
	E_OCV_DONE:

		(* update outputs *)
		bDone := TRUE;
		bBusy := FALSE;

		eState := E_OCV_IDLE;


(* unknown state *)
ELSE

	eState := E_OCV_IDLE;

	(* clear outputs *)
	bDone := FALSE;
	bBusy := FALSE;
	bError := FALSE;
	nErrorID := 0;
	strLastOCVFile := '';
	bOCVFileFound := FALSE;
	bOCVFileValid := FALSE;
	strLastCode := '';
END_CASE

END_FUNCTION_BLOCK

// ---- POUs/_Exclude/v2/FB_CAC_MoveFromArchive.TcPOU
(* restores OAC files from OAC archive for strCaseBarcode *)
FUNCTION_BLOCK FB_CAC_MoveFromArchive
VAR_INPUT
	bExecute					: BOOL;			(* set TRUE to move CAC file from Archive to Restore folder *)
	bDatabaseConfigured		: BOOL;
	sCaseBarcode				: T_CASE_Barcode;	(* case barcode *)
	sLocalCACPath				: STRING(255);	(* local CAC folder *)
	sLocalDbRestoreCACPath		: STRING(255);	(* local CAC folder *)
	stSystemTime				: TIMESTRUCT;	(* system time *)
	sRSKU					: T_CodeRSKU;
	sProductionOrder			: T_CodePO;
END_VAR
VAR_IN_OUT
	stCodeInfo_Case			: ST_CodeInfo;
END_VAR
VAR_OUTPUT
	bDone 					: BOOL;		(* TRUE = CAC restore complete *)
	bBusy 					: BOOL;		(* TRUE = CAC restore active *)
	bError 					: BOOL;		(* TRUE = CAC restore error *)
	nErrorID					: UDINT;	(* error code *)
	bCACFileFound				: BOOL;
	sCACFile					: T_CAC_Filename;
END_VAR
VAR
	fbExecute					: R_TRIG;
	eState					: E_CAC_State;
	eErrorState				: E_CAC_State;

	sSerialCode				: STRING;
	sDateFolder				: STRING(9);
	fbFindFile					: FB_EnumFindFileEntry;
	fbMoveFile				: FB_FileRename;
	eCmd 					: E_EnumCmdType;
	sPOFromCaseLabel			: T_CodePO;
	sRSKUFromCaseLabel		: T_CodeRSKU;
	sRSKUFromCaseLabel_test		: T_CodeRSKU;

END_VAR

fbExecute(CLK := bExecute);

CASE eState OF

	(* idle *)
	E_CAC_IDLE:

		(* restore file *)
		IF fbExecute.Q = TRUE THEN

			(* update outputs *)
			bDone := FALSE;
			bBusy := TRUE;
			bError := FALSE;
			nErrorID := 0;
			eErrorState := eState;

			(* convert sCaseBarcode to CAC Filename and extract date *)
			bCACFileFound := FALSE;

			sPOFromCaseLabel := F_CODE_GetItem(sCaseBarcode, eCodeAIType.ProductionOrder, stCodeInfo_Case);
			sRSKUFromCaseLabel := F_CODE_GetItem(sCaseBarcode, eCodeAIType.RSKU, stCodeInfo_Case);

			sRSKUFromCaseLabel_test := F_CASE_GetSKUFromHex( sRSKUFromCaseLabel) ;

			sCACFile := F_CONCAT3('CAC_', F_CASE_BarcodeToCACFilename(sCaseBarcode, stSystemTime, FALSE), '.xml');

			IF stCodeInfo_Case.stProductionOrder.nListPosition = 0 AND
				((  LEN(sRSKUFromCaseLabel) = 7 AND
					sRSKU = F_CASE_GetSKUFromHex( sRSKUFromCaseLabel))	OR
				(  LEN(sRSKUFromCaseLabel) > 7 AND
					sRSKU =  sRSKUFromCaseLabel) ) 	THEN

					sDateFolder := sRSKU;

			ELSIF sPOFromCaseLabel <> ''  						AND
				LEN(sPOFromCaseLabel) = LEN(sProductionOrder)	AND
				sRSKUFromCaseLabel = sRSKU						THEN

				sDateFolder := sPOFromCaseLabel;

			ELSIF sProductionOrder  <> '' THEN

				sDateFolder := sProductionOrder;
			ELSE
				sDateFolder := F_SYSTEM_SystemTimeToFolderName(stSystemTime);
			END_IF

			eCmd := eEnumCmd_First;

			eState := E_CAC_FINDFILE;

		(* bExecute has been reset *)
		ELSIF bExecute = FALSE THEN

			(* clear outputs *)
			bDone := FALSE;
			bBusy := FALSE;
			bError := FALSE;
			nErrorID := 0;
		END_IF


	(* find CAC file *)
	E_CAC_FINDFILE:

		(* find file *)
		fbFindFile(
			sNetId		:= '',
			sPathName	:= F_CONCAT5(sLocalCACPath, 'Archive\', sDateFolder, '\', sCACFile),
			eCmd		:= eCmd,
			bExecute	:= TRUE,
			tTimeout	:= T#1s
		);

		(* find file complete *)
		IF fbFindFile.bBusy = FALSE THEN

			(* find file completed OK *)
			IF fbFindFile.bError = FALSE THEN

				(* end of list *)
				IF fbFindFile.bEOE = TRUE THEN

					eState := E_CAC_DONE;

				(* file found *)
				ELSE

					(* log filename and update eCmd for next pass *)
					bCACFileFound := TRUE;
					sCACFile := fbFindFile.stFindFile.sFileName;
					eCmd := eEnumCmd_Next;

					eState := E_CAC_MOVEFILE;
				END_IF

			(* find file error *)
			ELSE

				bError := TRUE;
				nErrorID := fbFindFile.nErrID;
				eErrorState := eState;

				eState := E_CAC_DONE;
			END_IF


			(* close off fbFindFile *)
			fbFindFile(bExecute := FALSE);
		END_IF


	(* move CAC file from archive to CAC watch folder *)
	E_CAC_MOVEFILE:

		(* move file *)
	IF bDatabaseConfigured THEN
		fbMoveFile(
			sNetId	:= '',
			sOldName:= F_CONCAT5(sLocalCACPath, 'Archive\', sDateFolder, '\', sCACFile),
			sNewName:=CONCAT(sLocalDbRestoreCACPath,  sCACFile),
			ePath	:= PATH_GENERIC,
			bExecute:= TRUE,
			tTimeout:= T#1s
		);
	ELSE
		fbMoveFile(
			sNetId	:= '',
			sOldName:= F_CONCAT5(sLocalCACPath, 'Archive\', sDateFolder, '\', sCACFile),
			sNewName:=  F_CONCAT3(sLocalCACPath, 'Restore\', sCACFile),
			ePath	:= PATH_GENERIC,
			bExecute:= TRUE,
			tTimeout:= T#1s
		);
	END_IF

		(* move file complete *)
		IF fbMoveFile.bBusy = FALSE THEN

			(* move file completed OK *)
			IF fbMoveFile.bError = FALSE THEN

				eState := E_CAC_DONE;

			(* move file error *)
			ELSE

				bError := TRUE;
				nErrorID := fbMoveFile.nErrId;
				eErrorState := eState;
			END_IF

			eState := E_CAC_FINDFILE;

			(* close off fbMoveFile *)
			fbMoveFile(bExecute := FALSE);
		END_IF


	(* complete *)
	E_CAC_DONE:

		(* update outputs *)
		bBusy := FALSE;
		bDone := TRUE;

		eState := E_CAC_IDLE;

(* unknoen state *)
ELSE

	eState := E_CAC_IDLE;
END_CASE

END_FUNCTION_BLOCK

// ---- POUs/_Exclude/F41_EventLoggerPT.TcPOU
PROGRAM F41_EventLoggerPT
VAR
	fbLogEventTime			: NT_GetTime;
	fbSystemTime				: RTC_EX2;
	rtWriteLogData				: R_TRIG;

	nImageByte				: UINT;
	(*aDataLogImage				: ARRAY[0..65000] OF BYTE;*)
	fbWriteFile				: FB_FILE_ApendWriteByByte;

	sCurrentLogPathFile			: STRING;
	sMemoLogPathFile				: STRING;
END_VAR

IF NOT stMachineConfig.bSystemLogEnable THEN
	MEMSET(ADR(gProcess.stEventDataPT.aDataLogImage), 16#00, SIZEOF(gProcess.stEventDataPT.aDataLogImage));
	MEMSET(ADR(stWriteImageData.aLogPT), 16#00, SIZEOF(stWriteImageData.aLogPT));
	gProcess.stEventDataPT.bEnable		:= FALSE;
	RETURN;
ELSE
	gProcess.stEventDataPT.bEnable := stMetsStatus.bSystemTimeValid;
END_IF



(* 	$T - Tab
	$R$N - end line + carier return*)
(*sCurrentLogPathFile	:= F_CONCAT6(stMetsStatus.sLocalSystemLog,'DL_',F_SYSTEM_Date(fbSystemTime.CDT),'_', LEFT(F_SYSTEM_TimeSuperFine(fbSystemTime.CDT),2), '.txt');*)
sCurrentLogPathFile	:= F_CONCAT4(stMetsStatus.sLocalSystemLogPath,'METS-PT_',F_SYSTEM_Date(stMetsStatus.stCTDateTime.sSystemTime), '.txt');

(*stEventData.sTimeStamp := F_SYSTEM_SystemTimeAsISO8601(fbSystemTime.CDT, stMetsStatus.stCTDateTime.sUTCTimeZoneOffset );*)
gProcess.stEventDataPT.sTimeStamp :=MID( F_SYSTEM_SystemTimeAsISO8601(stMetsStatus.stCTDateTime.sSystemTime, stMetsStatus.stCTDateTime.sUTCTimeZoneOffset ), 12, 12);

rtWriteLogData(CLK:= bPulse1s AND gProcess.stEventDataPT.bEnable);

IF rtWriteLogData.Q THEN
	MEMMOVE(ADR(stWriteImageData.aLogPT), ADR(gProcess.stEventDataPT.aDataLogImage), SIZEOF(gProcess.stEventDataPT.aDataLogImage));
	nImageByte := gProcess.stEventDataPT.nImageByte;

	IF sCurrentLogPathFile <> sMemoLogPathFile THEN
		gProcess.stEventDataPT.nCounter :=0;
		sMemoLogPathFile := sCurrentLogPathFile;
	END_IF

END_IF

fbWriteFile(
	bExecute	:= rtWriteLogData.Q AND nImageByte <> 0,
	pSourceAddr	:= ADR(stWriteImageData.aLogPT),
	nSourceSize	:= nImageByte,
	strPathFile	:= sCurrentLogPathFile,
	tTimeout	:= T#1s
);

IF rtWriteLogData.Q  THEN


	gProcess.stEventDataPT.bBufferOverflow := FALSE;
	gProcess.stEventDataPT.nImageByte := 0;
	gProcess.stEventDataPT.nControlSize := 0;
	MEMSET(ADR(gProcess.stEventDataPT.aDataLogImage), 16#00, SIZEOF(gProcess.stEventDataPT.aDataLogImage));

END_IF

END_PROGRAM

// ---- POUs/_Exclude/F42_EventLoggerML.TcPOU
PROGRAM F42_EventLoggerML
VAR
	fbLogEventTime			: NT_GetTime;
	fbSystemTime				: RTC_EX2;
	rtWriteLogData				: R_TRIG;

	nImageByte				: UINT;
	(*aDataLogImage				: ARRAY[0..65000] OF BYTE;*)
	fbWriteFile				: FB_FILE_ApendWriteByByte;

	sCurrentLogPathFile			: STRING;
	sMemoLogPathFile				: STRING;
END_VAR

IF NOT stMachineConfig.bSystemLogEnable THEN
	MEMSET(ADR(gProcess.stEventDataML.aDataLogImage), 16#00, SIZEOF(gProcess.stEventDataML.aDataLogImage));
	MEMSET(ADR(stWriteImageData.aLogML), 16#00, SIZEOF(stWriteImageData.aLogML));
	gProcess.stEventDataML.bEnable	:= FALSE;
	RETURN;
ELSE
	gProcess.stEventDataML.bEnable := stMetsStatus.bSystemTimeValid;
END_IF


(* 	$T - Tab
	$R$N - end line + carier return*)
(*sCurrentLogPathFile	:= F_CONCAT6(stMetsStatus.sLocalSystemLog,'DL_',F_SYSTEM_Date(fbSystemTime.CDT),'_', LEFT(F_SYSTEM_TimeSuperFine(fbSystemTime.CDT),2), '.txt');*)
sCurrentLogPathFile	:= F_CONCAT4(stMetsStatus.sLocalSystemLogPath,'METS-ML_',F_SYSTEM_Date(stMetsStatus.stCTDateTime.sSystemTime), '.txt');

(*stEventData.sTimeStamp := F_SYSTEM_SystemTimeAsISO8601(fbSystemTime.CDT, stMetsStatus.stCTDateTime.sUTCTimeZoneOffset );*)
gProcess.stEventDataML.sTimeStamp :=MID( F_SYSTEM_SystemTimeAsISO8601(stMetsStatus.stCTDateTime.sSystemTime, stMetsStatus.stCTDateTime.sUTCTimeZoneOffset ), 12, 12);

rtWriteLogData(CLK:= bPulse10s AND gProcess.stEventDataML.bEnable);

IF rtWriteLogData.Q THEN
	MEMMOVE(ADR(stWriteImageData.aLogML), ADR(gProcess.stEventDataML.aDataLogImage), SIZEOF(gProcess.stEventDataML.aDataLogImage));
	nImageByte := gProcess.stEventDataML.nImageByte;

	IF sCurrentLogPathFile <> sMemoLogPathFile THEN
		gProcess.stEventDataML.nCounter :=0;
		sMemoLogPathFile := sCurrentLogPathFile;
	END_IF

END_IF

fbWriteFile(
	bExecute	:= rtWriteLogData.Q AND nImageByte <> 0, (*AND nLogSeq < 5*)
	pSourceAddr	:= ADR(stWriteImageData.aLogML),
	nSourceSize	:= nImageByte,
	strPathFile	:= sCurrentLogPathFile,(*F_CONCAT6(stMetsStatus.sLocalSystemLog,'DL_',F_SYSTEM_Date(fbSystemTime.CDT),'_', LEFT(F_SYSTEM_TimeSuperFine(fbSystemTime.CDT),2), '.txt'),*)
	tTimeout	:= T#1s
);

IF rtWriteLogData.Q  (*AND nLogSeq < 5*) THEN

	(*nLogSeq  := nLogSeq +1;*)
	gProcess.stEventDataML.bBufferOverflow := FALSE;
	gProcess.stEventDataML.nImageByte := 0;
	gProcess.stEventDataML.nControlSize := 0;
	MEMSET(ADR(gProcess.stEventDataML.aDataLogImage), 16#00, SIZEOF(gProcess.stEventDataML.aDataLogImage));

END_IF

END_PROGRAM

// ---- POUs/_Exclude/F43_EventLoggerOT.TcPOU
PROGRAM F43_EventLoggerOT
VAR
	fbLogEventTime			: NT_GetTime;
	fbSystemTime				: RTC_EX2;
	rtWriteLogData				: R_TRIG;

	nImageByte				: UINT;
	(*aDataLogImage				: ARRAY[0..65000] OF BYTE;*)
	fbWriteFile				: FB_FILE_ApendWriteByByte;

	sCurrentLogPathFile			: STRING;
	sMemoLogPathFile				: STRING;
END_VAR

IF NOT stMachineConfig.bSystemLogEnable THEN
	MEMSET(ADR(gProcess.stEventDataOT.aDataLogImage), 16#00, SIZEOF(gProcess.stEventDataOT.aDataLogImage));
	MEMSET(ADR(stWriteImageData.aLogOT), 16#00, SIZEOF(stWriteImageData.aLogOT));
	gProcess.stEventDataOT.bEnable		:= FALSE;
	RETURN;
ELSE
	gProcess.stEventDataOT.bEnable := stMetsStatus.bSystemTimeValid;
END_IF



(* 	$T - Tab
	$R$N - end line + carier return*)
(*sCurrentLogPathFile	:= F_CONCAT6(stMetsStatus.sLocalSystemLog,'DL_',F_SYSTEM_Date(fbSystemTime.CDT),'_', LEFT(F_SYSTEM_TimeSuperFine(fbSystemTime.CDT),2), '.txt');*)
sCurrentLogPathFile	:= F_CONCAT4(stMetsStatus.sLocalSystemLogPath,'METS-OT_',F_SYSTEM_Date(stMetsStatus.stCTDateTime.sSystemTime), '.txt');

(*stEventData.sTimeStamp := F_SYSTEM_SystemTimeAsISO8601(fbSystemTime.CDT, stMetsStatus.stCTDateTime.sUTCTimeZoneOffset );*)
gProcess.stEventDataOT.sTimeStamp :=MID( F_SYSTEM_SystemTimeAsISO8601(stMetsStatus.stCTDateTime.sSystemTime, stMetsStatus.stCTDateTime.sUTCTimeZoneOffset ), 12, 12);

rtWriteLogData(CLK:= bPulse1s AND gProcess.stEventDataOT.bEnable);

IF rtWriteLogData.Q THEN
	MEMMOVE(ADR(stWriteImageData.aLogOT), ADR(gProcess.stEventDataOT.aDataLogImage), SIZEOF(gProcess.stEventDataOT.aDataLogImage));
	nImageByte := gProcess.stEventDataOT.nImageByte;

	IF sCurrentLogPathFile <> sMemoLogPathFile THEN
		gProcess.stEventDataOT.nCounter :=0;
		sMemoLogPathFile := sCurrentLogPathFile;
	END_IF

END_IF

fbWriteFile(
	bExecute	:= rtWriteLogData.Q AND nImageByte <> 0,
	pSourceAddr	:= ADR(stWriteImageData.aLogOT),
	nSourceSize	:= nImageByte,
	strPathFile	:= sCurrentLogPathFile,
	tTimeout	:= T#1s
);

IF rtWriteLogData.Q  THEN


	gProcess.stEventDataOT.bBufferOverflow := FALSE;
	gProcess.stEventDataOT.nImageByte := 0;
	gProcess.stEventDataOT.nControlSize := 0;
	MEMSET(ADR(gProcess.stEventDataOT.aDataLogImage), 16#00, SIZEOF(gProcess.stEventDataOT.aDataLogImage));

END_IF

END_PROGRAM

// ---- POUs/_Exclude/F44_EventLoggerCT.TcPOU
PROGRAM F44_EventLoggerCT
VAR
	fbLogEventTime			: NT_GetTime;
	fbSystemTime				: RTC_EX2;
	rtWriteLogData				: R_TRIG;

	nImageByte				: UINT;
	aDataLogImage				: ARRAY[0..65000] OF BYTE;
	fbWriteFile				: FB_FILE_ApendWriteByByte;

	sCurrentLogPathFile			: STRING;
	sMemoLogPathFile				: STRING;
END_VAR

IF NOT stMachineConfig.bSystemLogEnable THEN
	MEMSET(ADR(gProcess.stEventDataCT.aDataLogImage), 16#00, SIZEOF(gProcess.stEventDataCT.aDataLogImage));
	MEMSET(ADR(stWriteImageData.aLogCT), 16#00, SIZEOF(stWriteImageData.aLogCT));
	gProcess.stEventDataCT.bEnable	:= FALSE;
	RETURN;
ELSE
	gProcess.stEventDataCT.bEnable := stMetsStatus.bSystemTimeValid;
END_IF


(* 	$T - Tab
	$R$N - end line + carier return*)
(*sCurrentLogPathFile	:= F_CONCAT6(stMetsStatus.sLocalSystemLog,'DL_',F_SYSTEM_Date(fbSystemTime.CDT),'_', LEFT(F_SYSTEM_TimeSuperFine(fbSystemTime.CDT),2), '.txt');*)
sCurrentLogPathFile	:= F_CONCAT4(stMetsStatus.sLocalSystemLogPath,'METS-CT_',F_SYSTEM_Date(stMetsStatus.stCTDateTime.sSystemTime), '.txt');

(*stEventData.sTimeStamp := F_SYSTEM_SystemTimeAsISO8601(fbSystemTime.CDT, stMetsStatus.stCTDateTime.sUTCTimeZoneOffset );*)
gProcess.stEventDataCT.sTimeStamp :=MID( F_SYSTEM_SystemTimeAsISO8601(stMetsStatus.stCTDateTime.sSystemTime, stMetsStatus.stCTDateTime.sUTCTimeZoneOffset ), 12, 12);

rtWriteLogData(CLK:= bPulse1s AND gProcess.stEventDataCT.bEnable);

IF rtWriteLogData.Q THEN
	MEMMOVE(ADR(stWriteImageData.aLogCT), ADR(gProcess.stEventDataCT.aDataLogImage), SIZEOF(gProcess.stEventDataCT.aDataLogImage));
	nImageByte := gProcess.stEventDataCT.nImageByte;

	IF sCurrentLogPathFile <> sMemoLogPathFile THEN
		gProcess.stEventDataCT.nCounter :=0;
		sMemoLogPathFile := sCurrentLogPathFile;
	END_IF

END_IF

fbWriteFile(
	bExecute	:= rtWriteLogData.Q AND nImageByte <> 0, (*AND nLogSeq < 5*)
	pSourceAddr	:= ADR(stWriteImageData.aLogCT),
	nSourceSize	:= nImageByte,
	strPathFile	:= sCurrentLogPathFile,(*F_CONCAT6(stMetsStatus.sLocalSystemLog,'DL_',F_SYSTEM_Date(fbSystemTime.CDT),'_', LEFT(F_SYSTEM_TimeSuperFine(fbSystemTime.CDT),2), '.txt'),*)
	tTimeout	:= T#1s
);

IF rtWriteLogData.Q  (*AND nLogSeq < 5*) THEN

	(*nLogSeq  := nLogSeq +1;*)
	gProcess.stEventDataCT.bBufferOverflow := FALSE;
	gProcess.stEventDataCT.nImageByte := 0;
	gProcess.stEventDataCT.nControlSize := 0;
	MEMSET(ADR(gProcess.stEventDataCT.aDataLogImage), 16#00, SIZEOF(gProcess.stEventDataCT.aDataLogImage));

END_IF

END_PROGRAM

// ---- POUs/_Exclude/FB_CASE_AddOACDataLoop.TcPOU
FUNCTION_BLOCK FB_CASE_AddOACDataLoop
VAR_INPUT
	bExecute					: BOOL;			(* scan for valid Outer in arrOuterStatus *)
	bStopOnInvalidCode		: BOOL;						(* set TRUE to give alarm if an invalid code is detected *)
	bFileReadOnly				: BOOL;
	bATTPModeEnable			: BOOL;
	sLocalOACPath				: STRING(50);	(* TEMP folder path *)
	stCTDateTime				: ST_SYSTEM_DateTime;	(* CaseTrace date/time structure *)
	stOuterDataNotFound		: ST_RejectItems;
END_VAR
VAR_IN_OUT
	stProductInstruction			: ST_PCM_Status;
	aOuterStatus				: ARRAY[1..cMAX_OUTER_STATUS_QUEUE] OF ST_OUTER_Status;	(* Outer status array *)
	stInfeedQueue				: ST_CASE_InfeedQueue;	(* Infeed Conveyor queue *)
END_VAR
VAR_OUTPUT
	bDone					: BOOL;			(* TRUE = write OAC file complete *)
	bBusy					: BOOL;			(* TRUE = write OAC file in progress *)
	bError					: BOOL;			(* TRUE = write OAC file error *)
	nErrorID					: UDINT;			(* error ID *)

	nOACFilesRead				: UDINT;
	nReadOACDataFromStructure	: INT;
	nReadOACDataFromFile		: INT;
	nOACFilesFalseRead 		: INT;

	sOACFile					: T_OAC_Filename;
	stOACData				: ST_OAC_Data;
	bScaningActive			: BOOL;
END_VAR
VAR
	fbExecute					: R_TRIG;
	eState					: E_CASE_State;
	eErrorState				: E_CASE_State;
	nOuterIndex				: INT;
	nMaxOuterIndex			: INT;

	sCurrnetInfeedBarcode		: T_MaxString;
	fbReadXMLData			: FB_XmlSrvRead;
	nScanIndex				: INT;

	sOuterTimeStamp				: T_ISO8601Time;
	bOuterMasterListRestored	: BOOL;
	sDataSource				: STRING(4);

	nCounter					: INT;
END_VAR

(* monitor bExecute for rising edge *)
fbExecute(CLK := bExecute);

CASE eState OF

	(* idle state *)
	E_CASE_IDLE:

		(* rising edge of bExecute *)
		IF fbExecute.Q = TRUE THEN

			(* update outputs *)
			bDone := FALSE;
			bBusy := TRUE;
			bError := FALSE;
			nErrorID := 0;

			(* clear outputs *)
			nOACFilesRead := 0;
			sOACFile := '';
			(*MEMSET(ADR(stOACData), 16#00, SIZEOF(stOACData));*)
			sDataSource :='';
			nMaxOuterIndex := UDINT_TO_INT(SIZEOF(aOuterStatus) / SIZEOF(aOuterStatus[1]));

			(*nOuterIndex := 1;*)

			eState := E_CASE_SCANINFEEDQUEUE;

		(* OAC data disabled *)
		ELSIF bExecute = FALSE THEN

			(* reset outputs *)
			bDone := FALSE;
			bBusy := FALSE;
			bError := FALSE;
			nErrorID := 0;

			bScaningActive := FALSE;

		END_IF


	(* scan for missing OAC data *)
	E_CASE_SCANINFEEDQUEUE:

		(* preset next state, will be udpated if an Outer without OAC data is found in Infeed Queue *)
		MEMSET(ADR(stOACData), 16#00, SIZEOF(stOACData));
		eState := E_CASE_DONE;

		(* scan remainder of Infeed Queue *)
		FOR nScanIndex := 1 TO  MIN(stInfeedQueue.nIndex, cMAX_INFEED_QUEUE) DO

			(* OAC data has not been read *)
			IF stInfeedQueue.aOuter[nScanIndex].CodingAndTrackingMode = 0 AND  stInfeedQueue.aOuter[nScanIndex].DataSource = '' THEN

				IF (*stProductInstruction.nOpMode = 7 AND*) NOT stProductInstruction.bEnablePacks (*AND bStopOnInvalidCode*) THEN
					stInfeedQueue.aOuter[nScanIndex].ProductionDate := F_StringWildcard('#YYYYMMDD#', stCTDateTime.sSystemTime);
					stInfeedQueue.aOuter[nScanIndex].ProductionTime := F_StringWildcard('#hhmmss#', stCTDateTime.sSystemTime);
					stInfeedQueue.aOuter[nScanIndex].ProductionTimeOffset := F_SYSTEM_SystemTimeOffsetToHHMM(stCTDateTime.nSystemTimeOffset);

					stInfeedQueue.aOuter[nScanIndex].OuterTimeStamp :=F_SYSTEM_SystemTimeAsISO8601(stCTDateTime.sSystemTime, stCTDateTime.sUTCTimeZoneOffset );
					stInfeedQueue.aOuter[nScanIndex].RetailSKU := stProductInstruction.sRetailSKU;
					stInfeedQueue.aOuter[nScanIndex].OuterMachine.ProductionSite :=  stProductInstruction.sProductionSite;
					stInfeedQueue.aOuter[nScanIndex].OuterMachine.ProductionLine := stProductInstruction.sProductionLine;
					stInfeedQueue.aOuter[nScanIndex].BatchNumber := stProductInstruction.sBatchNumber;
					stInfeedQueue.aOuter[nScanIndex].CodingAndTrackingMode := stProductInstruction.nOpMode;

					stInfeedQueue.aOuter[nScanIndex].DataSource := 'REST';
					stInfeedQueue.aOuter[nScanIndex].OuterRejectCode := 'OK';
					stInfeedQueue.aOuter[nScanIndex].OuterRejectID := 0;

					eState := E_CASE_SCANINFEEDQUEUE;

				ELSE
					sCurrnetInfeedBarcode 	:=	 stInfeedQueue.aOuter[nScanIndex].Barcode ;
					bOuterMasterListRestored 	:= stInfeedQueue.aOuter[nScanIndex].OuterMasterListRestored;
					(*sOuterTimeStamp			:= stInfeedQueue.aOuter[nScanIndex].OuterTimeStamp;*)
					sDataSource :='';
					(* generate OAC file name and clear data for last OAC file *)

					sOACFile := F_CONCAT3('OAC_', F_OUTER_BarcodeToHex(sCurrnetInfeedBarcode), '.xml');

					IF bFileReadOnly THEN
						eState := E_CASE_READOACDATA;
					ELSE
						eState := E_CASE_SCANOUTERS;
					END_IF
				END_IF

				bScaningActive := TRUE;
				EXIT;
			END_IF
		END_FOR

	E_CASE_SCANOUTERS:


		FOR nOuterIndex := 1 TO nMaxOuterIndex DO

			(* TriggerID > 0 indicates Outer data present *)
			IF aOuterStatus[nOuterIndex].bLabelApplied AND
				 NOT aOuterStatus[nOuterIndex].nStatus.19 AND
				NOT aOuterStatus[nOuterIndex].nStatus.22 THEN

				IF  aOuterStatus[nOuterIndex].stOACData.Barcode = sCurrnetInfeedBarcode THEN

					stOACData	 := aOuterStatus[nOuterIndex].stOACData;
					EXIT;
				END_IF
			END_IF
		END_FOR

		IF stOACData.CodingAndTrackingMode > 0 OR stOACData.OuterRejectCode <> '' THEN

			nOACFilesRead := nOACFilesRead + 1;
			sDataSource := 'ST';
			nReadOACDataFromStructure:= nReadOACDataFromStructure + 1;

			eState := E_CASE_UPDATEINFEEDQUEUE;
		ELSE
			eState := E_CASE_READOACDATA;
		END_IF

	(* read data from OAC *)
	E_CASE_READOACDATA:

(* read data using XML Server *)
		fbReadXMLData(
			sNetId		:= '',
			ePath		:= PATH_GENERIC,
			nMode		:= XMLSRV_SKIPMISSING,
			pSymAddr	:= ADR(stOACData),
			cbSymSize	:= SIZEOF(stOACData),
			sFilePath		:= CONCAT(sLocalOACPath, sOACFile),
			sXPath		:= '/Outer',
			bExecute		:= TRUE,
			tTimeout		:= T#1s
		);
		(* file read complete *)
		IF fbReadXMLData.bBusy = FALSE THEN

			(* file read completed OK *)
			IF fbReadXMLData.bError = FALSE THEN

				(* update counter *)
				nOACFilesRead := nOACFilesRead + 1;
				nReadOACDataFromFile:= nReadOACDataFromFile + 1;
				sDataSource := 'FILE';

			(* file read error *)
			ELSE

				bError := TRUE;
				nErrorID := fbReadXMLData.nErrId;
				nOACFilesFalseRead := nOACFilesFalseRead + 1;
				sDataSource := 'NO_R';

				stOACData.OuterRejectCode 	:= stOuterDataNotFound.sMetsDisplayCode;
				stOACData.OuterRejectID		:= stOuterDataNotFound.nRejectID;
				eErrorState := eState;
			END_IF

			eState := E_CASE_UPDATEINFEEDQUEUE;

			(* close off fbReadXMLData *)
			fbReadXMLData(bExecute := FALSE);
		END_IF

	(* update OAC data to Infeed Queue *)
	E_CASE_UPDATEINFEEDQUEUE:

		(* scan Infeed Queue *)
		FOR nScanIndex := 1 TO  MIN(stInfeedQueue.nIndex, cMAX_INFEED_QUEUE) DO

			(* generate OAC file name AND clear data FOR last OAC file *)
				(* Outer is still in same position in Infeed Queue *)
			IF stInfeedQueue.aOuter[nScanIndex].Barcode = sCurrnetInfeedBarcode THEN

				(* copy OAC data into Infeed Queue *)
				IF stOACData.Barcode = sCurrnetInfeedBarcode AND  stOACData.Barcode <> '' THEN
					stInfeedQueue.aOuter[nScanIndex] := stOACData;
				(*In case File read return error and erase stOACData*)
				ELSIF stOACData.Barcode ='' THEN
					stInfeedQueue.aOuter[nScanIndex].Barcode := sCurrnetInfeedBarcode;
				ELSE
					stInfeedQueue.aOuter[nScanIndex].Barcode := sCurrnetInfeedBarcode;
					stInfeedQueue.aOuter[nScanIndex].DataSource := 'MISS';
				END_IF
				(*stInfeedQueue.aOuter[nScanIndex].OuterTimeStamp			:= sOuterTimeStamp;*)
				stInfeedQueue.aOuter[nScanIndex].DataSource 				:= sDataSource;
				stInfeedQueue.aOuter[nScanIndex].OuterMasterListRestored 	:= bOuterMasterListRestored;
				stInfeedQueue.aOuter[nScanIndex].OuterCodeStatus.4 		:= bOuterMasterListRestored;

				(*Modif outer time stamp to represent moment of adding OCA data in casepacker*)
				IF bATTPModeEnable THEN
					stInfeedQueue.aOuter[nScanIndex].OuterTimeStamp :=F_SYSTEM_SystemTimeAsISO8601(stCTDateTime.sSystemTime, stCTDateTime.sUTCTimeZoneOffset );
				END_IF

				EXIT;
			END_IF
		END_FOR

		eState := E_CASE_SCANINFEEDQUEUE;

	(* done *)
	E_CASE_DONE:

		bScaningActive := FALSE;

		(* update outputs *)
		bBusy := FALSE;
		bDone := TRUE;

		eState := E_CASE_IDLE;


(* unknown state *)
ELSE

	eState := E_CASE_IDLE;
END_CASE

END_FUNCTION_BLOCK

// ---- POUs/_Exclude/FB_CASE_ShiftCaseQueue_ORG.TcPOU
(* shifts specified group of cases in CaseQueue by 1 index *)
FUNCTION_BLOCK FB_CASE_ShiftCaseQueue_ORG
VAR_INPUT
	bExecute					: BOOL;			(* set TRUE to shift Case Queue *)
	bLogCaseOwerwriten		: BOOL;
	stCTDateTime				: ST_SYSTEM_DateTime;
	nFirstCaseIndex			: INT;			(* index of 1st case to be shifted *)
	nLastCaseIndex			: INT;			(* index of last case position owerwriten *)
	bStopOnOverWrittenData	: BOOL;
	tTimeOut					: TIME;
END_VAR
VAR_IN_OUT
	stCaseQueue				: ST_CASE_CaseQueue;	(* Case Queue *)
	stCaseQueueHMI			: ST_HMI_CASE_CaseQueue;	(* Case Queue *)
	(*bFoundNotEmptyTarget		: BOOL;*)
END_VAR
VAR_OUTPUT
	bDone					: BOOL;			(* TRUE = complete *)
	bBusy					: BOOL;
	bError					: BOOL;			(* TRUE = nFirstIndex and nLastCaseIndex not valid *)
	nErrorID					: UDINT;
	bFoundNotEmptyTarget		: BOOL;
END_VAR
VAR
	fbExecute					: R_TRIG;
	nMaxCaseIndex			: INT;

	eStep					: E_CASE_State;
	eErrorState				: E_CASE_State;

	tonTimeOut					:	TON;

	stCACDataToLog					:  ST_CAC_Data;	(* array of CAC data *)
	nCaseQueueToShift				: INT;
	bLogOwerwritenDataToFileEx		: BOOL;
	fbLogOwerwritenCACData		: FB_CAC_WriteFile;

END_VAR

(* rising edge of bExecute *)
fbExecute(CLK:= bExecute);

tonTimeOut(IN:= eStep=E_CASE_DATAWRITEXML, PT:= tTimeOut);

CASE eStep OF

	E_CASE_IDLE:
		(* move CaseData *)
		IF fbExecute.Q = TRUE THEN

			bDone := FALSE;
			bBusy := TRUE;
			bError := FALSE;
			nErrorID	:= 0;
	
			eErrorState	:=eStep;
			(* max index of Case Queue buffer *)
			nMaxCaseIndex := UDINT_TO_INT(SIZEOF(stCaseQueue.aCACData) / SIZEOF(stCaseQueue.aCACData[1]));
			bFoundNotEmptyTarget := FALSE;
			bLogOwerwritenDataToFileEx	:= FALSE;
			 MEMSET(ADR(stCACDataToLog), 16#00, SIZEOF(stCACDataToLog));
			(*nLastCaseIndex := nFirstCaseIndex + nTotalCasesToShift ;*)
			eStep :=E_CASE_DATAVALIDATE;
	
		(* bExecute has been reset *)
		ELSIF bExecute = FALSE THEN
	
			bDone := FALSE;
			bBusy := FALSE;
			bError := FALSE;
			nErrorID	:= 0;

			bFoundNotEmptyTarget := FALSE;
	
		END_IF

	E_CASE_DATAVALIDATE:
		(* specified range within buffer limits *)
		IF nFirstCaseIndex > 0 AND nLastCaseIndex <= nMaxCaseIndex THEN

			nCaseQueueToShift := nLastCaseIndex-nFirstCaseIndex;
			(* cases to be shifted > 0 *)
			IF  nCaseQueueToShift > 0 THEN

				stCACDataToLog	:= stCaseQueue.aCACData[MAX(1, nLastCaseIndex)];

				eStep :=E_CASE_DATAWRITEXML;

			ELSE
				bError := TRUE;
				eErrorState	:=eStep;
				nErrorID	:= 1;

				eStep :=E_CASE_DONE;
			END_IF
		(* nFirstIndex = 0 or specified range exceeds stCaseQueue limits *)
		ELSE
			bError := TRUE;
			eErrorState	:=eStep;
			nErrorID	:= 11;

			eStep :=E_CASE_DONE;
		END_IF

	E_CASE_DATAWRITEXML:

		IF stCaseQueue.aCACData[nLastCaseIndex].CodingAndTrackingMode <> 0 AND bLogCaseOwerwriten THEN

			bFoundNotEmptyTarget := bStopOnOverWrittenData;
			bLogOwerwritenDataToFileEx	:= TRUE;

			IF tonTimeOut.Q	THEN

				bError := TRUE;
				eErrorState	:=eStep;
				nErrorID	:= 2;

				eStep :=E_CASE_DATAFINALISE;


			ELSIF	 fbLogOwerwritenCACData.bDone THEN
				IF  fbLogOwerwritenCACData.bError THEN

					bError := TRUE;
					eErrorState	:=eStep;
					nErrorID	:= 22;
				END_IF

				eStep :=E_CASE_DATAFINALISE;
			END_IF
		ELSE
			eStep :=E_CASE_DATAFINALISE;
		END_IF

	E_CASE_DATAFINALISE:

		bLogOwerwritenDataToFileEx	:= FALSE;

		(* shift specified cases in CaseQueue *)
		MEMMOVE(ADR(stCaseQueue.aCACData[nFirstCaseIndex + 1]), ADR(stCaseQueue.aCACData[nFirstCaseIndex]), nCaseQueueToShift* SIZEOF(stCaseQueue.aCACData[1]));

		(* shift specified cases in CaseQueue *)
		MEMMOVE(ADR(stCaseQueueHMI.aCACData[nFirstCaseIndex + 1]), ADR(stCaseQueueHMI.aCACData[nFirstCaseIndex]), nCaseQueueToShift* SIZEOF(stCaseQueueHMI.aCACData[1]));

		(* clear data in 1st indexes *)
		MEMSET(ADR(stCaseQueue.aCACData[nFirstCaseIndex]), 16#00, SIZEOF(stCaseQueue.aCACData[nFirstCaseIndex]));

		(* clear data in 1st indexes *)
		MEMSET(ADR(stCaseQueueHMI.aCACData[nFirstCaseIndex]), 16#00, SIZEOF(stCaseQueueHMI.aCACData[nFirstCaseIndex]));

		eStep :=E_CASE_DONE;

	E_CASE_DONE:

		bFoundNotEmptyTarget := FALSE;

		bDone := TRUE;
		bBusy := FALSE;

		eStep :=E_CASE_IDLE;
ELSE
	eStep :=E_CASE_IDLE;
END_CASE

fbLogOwerwritenCACData(

(*Do zminany tak aby podawac finalna sciezke i inalna nazwe dla bloku WireFile_v2*)
	bExecute			:=	bLogOwerwritenDataToFileEx,
	bOverwrittenCAC	:= TRUE,
	strLocalCACPath	:= stMetsStatus.sLocalCACPath,
	strCaseFilename	:=F_CONCAT5('OVERWRITEN_Pos_',INT_TO_STRING(nLastCaseIndex),'_', F_SYSTEM_SystemTimeToCHM_Header(stCTDateTime.sSystemTime),'.xml'),
	stCACData			:= stCACDataToLog, (*stCaseQueue.stCACData[MAX(1, nLastCaseIndex)],*)
	bDone			=>,
	bBusy			=>,
	bError			=>,
	nErrorID			=>,
	bCACValid		=>,
	strCACFile		=>,
	strFirstOuter		=>,
	strLastOuter		=>
);

END_FUNCTION_BLOCK

// ---- POUs/_Exclude/v1/FB_CAC_WriteFile.TcPOU
FUNCTION_BLOCK FB_CAC_WriteFile
VAR_INPUT
	bExecute						: BOOL;
	bOverwrittenCAC					: BOOL;
	strLocalCACPath					: STRING(255);
	strLocalBridgePath					: STRING(255);
	bDataBaseConfigured				: BOOL;
	strCaseFilename				:STRING(255);
END_VAR
VAR_IN_OUT
	stCACData						: ST_CAC_Data;
END_VAR
VAR_OUTPUT
	bDone							: BOOL;
	bBusy							: BOOL;
	bError							: BOOL;
	nErrorID						: UDINT;
	bCACValid						: BOOL;
	strCACFile						: T_CAC_Filename;	(* CAC file name generated from stCACData *)
	strFirstOuter					: T_OUTER_Barcode;
	strLastOuter					: T_OUTER_Barcode;
	bBufferOverflow	: BOOL;
END_VAR
VAR
	fbExecute						: R_TRIG;
	eState							: E_CAC_State;
	eErrorState						: E_CAC_State;

	arrCACImage						: ARRAY[0..cMAX_FILE_BUFFER] OF BYTE;
	strString						: STRING(255);
	nStringLen						: INT;
	nCACByte						: UINT;
	nOuterIndex						: INT;
	nMaxCACImageSize	: UINT;
	nControlSize		: UINT;

	Debug	: UDINT;

	strTargetPath				 	: STRING(255);
	fbOpenFile						: FB_FileOpen;
	hFile							: UINT;
	fbCloseFile						: FB_FileClose;
	fbWriteFile						: FB_FileWrite;
	fbBuildOACData					: FB_OAC_BuildXMLData;
	fbPopulateMinimalOuterData			: FB_CAC_PopulateMinimalOuterData;
END_VAR

fbExecute(CLK := bExecute);

Debug := MAX(nCACByte, Debug);
CASE eState OF

	(* idle *)
	E_CAC_IDLE:

		IF fbExecute.Q = TRUE THEN

			(* update outputs *)
			bDone := FALSE;
			bBusy := TRUE;
			bError := FALSE;
			nErrorID := 0;

			(* initialise CAC byte and output image *)
			nCACByte := 0;
			MEMSET(ADR(arrCACImage), 16#00, SIZEOF(arrCACImage));
			nControlSize := 0;
			nMaxCACImageSize := SIZEOF(arrCACImage);


			(* build CAC template header fields *)
			(* XML header *)
			strString := cXML_HEADER;
			nStringLen := LEN(strString);
			MEMMOVE(ADR(arrCACImage[nCACByte]), ADR(strString), nStringLen);
			nCACByte := nCACByte + nStringLen;

			(* <Comment> tag *)
			strString := '<!--File CAC builder. Version 2.1.000 Relase 01.07.2021 PTR -->$R$N';
			AppendImageData();


			(* <Case> tag *)
			strString := '<Case>$R$N';
			AppendImageData();

			(* <Barcode> field *)
			strString := F_CONCAT3('$T<Barcode>', stCACData.Barcode, '</Barcode>$R$N');
			AppendImageData();

			(* <ProductionDate> field *)
			strString := F_CONCAT3('$T<ProductionDate>', stCACData.ProductionDate, '</ProductionDate>$R$N');
			AppendImageData();

			(* <ProductionTime> field *)
			strString := F_CONCAT3('$T<ProductionTime>', stCACData.ProductionTime, '</ProductionTime>$R$N');
			AppendImageData();

			(* <ProductionTimeOffset> field *)
			strString := F_CONCAT3('$T<ProductionTimeOffset>', stCACData.ProductionTimeOffset, '</ProductionTimeOffset>$R$N');
			AppendImageData();

			(* <RetailSKU> field *)
			strString := F_CONCAT3('$T<RetailSKU>', stCACData.RetailSKU, '</RetailSKU>$R$N');
			AppendImageData();

			(* <CasePacker> tag *)
			strString := '$T<CasePacker>$R$N';
			AppendImageData();

			(* <ProductionSite> field *)
			strString := F_CONCAT3('$T$T<ProductionSite>', stCACData.CasePacker.ProductionSite, '</ProductionSite>$R$N');
			AppendImageData();

			(* <ProductionLine> field *)
			strString := F_CONCAT3('$T$T<ProductionLine>', stCACData.CasePacker.ProductionLine, '</ProductionLine>$R$N');
			AppendImageData();

			(* </CasePacker> tag *)
			strString := '$T</CasePacker>$R$N';
			AppendImageData();

			(* <CodingAndTrackingMode> field *)
			strString := F_CONCAT3('$T<CodingAndTrackingMode>', INT_TO_STRING(stCACData.CodingAndTrackingMode), '</CodingAndTrackingMode>$R$N');
			AppendImageData();

			(* <NumberOfOuters> field *)
			strString := F_CONCAT3('$T<NumberOfOuters>', INT_TO_STRING(stCACData.NumberOfOuters), '</NumberOfOuters>$R$N');
			AppendImageData();

			(* generate CAC filename *)
			strCACFile := strCaseFilename;

			(* stCACData is valid *)
			IF F_ToUCase(stCACData.CaseRejectCode) = 'OK' AND NOT bOverwrittenCAC THEN

				(* write valid CAC files to TEMP folder *)
				bCACValid := TRUE;
				IF bDataBaseConfigured THEN
					strTargetPath := strLocalBridgePath;
				ELSE
					strTargetPath := strLocalCACPath;
				END_IF

				(* first and last Outers in CAC file *)
				strFirstOuter := stCACData.Outer[1].Barcode;
				strLastOuter := stCACData.Outer[stCACData.NumberOfOuters].Barcode;

			(* stCACData is invalid *)
			ELSE

				(* <CaseRejectCode> field *)
				strString := F_CONCAT3('$T<CaseRejectCode>', SEL(bOverwrittenCAC,  stCACData.CaseRejectCode, 'CACDataOver-written'), '</CaseRejectCode>$R$N');
				AppendImageData();


				(* <CaseRejectID> field *)
				strString := F_CONCAT3('$T<CaseRejectID>', UINT_TO_STRING(stCACData.CaseRejectID), '</CaseRejectID>$R$N');
				AppendImageData();

				(* generate CAC filename and target path for ErrCAC files *)
				bCACValid := FALSE;
				strCACFile := CONCAT('Err', strCACFile);
				strTargetPath := CONCAT(strLocalCACPath, 'Error\');

				(* reset first and last Outers *)
				strFirstOuter := '';
				strLastOuter := '';
			END_IF

			(* first Outer to be added to arrCACImage *)
			nOuterIndex := 1;

			eState := E_CAC_OPENFILE;

		(* bExecute has been reset *)
		ELSIF bExecute = FALSE THEN

			(* update outputs *)
			bDone := FALSE;
			bBusy := FALSE;
			bError := FALSE;
			nErrorID := 0;
		END_IF


	(* open CAC file for writing *)
	E_CAC_OPENFILE:

		fbOpenFile(
			sNetId		:= '',
			sPathName	:= CONCAT(strTargetPath, strCACFile),
			nMode		:= FOPEN_MODEWRITE OR FOPEN_MODEBINARY,
			ePath		:= PATH_GENERIC,
			bExecute	:= TRUE,
			tTimeout	:= T#1s
		);

		(* open file complete *)
		IF fbOpenFile.bBusy = FALSE THEN

			(* open file completed OK *)
			(*	OACdata now required in all modes	*)
			IF fbOpenFile.bError = FALSE THEN

				(* file handle *)
				hFile := fbOpenFile.hFile;

				(* OAC data required in CAC file *)
				IF stCACData.CodingAndTrackingMode >= 7 THEN

					eState := E_CAC_BUILDXMLIMAGE;

				(* OAC data not required in CAC file *)
				ELSE
					(* Fill in  Minimal data into stCACData.Outer*)
					fbPopulateMinimalOuterData(
					bExecute := TRUE,
					nNumberofOuters := stCACData.NumberOfOuters,
					stCACData := stCACData
					);

					IF fbPopulateMinimalOuterData.bDone THEN
						eState := E_CAC_BUILDXMLIMAGE;
					END_IF

(*
					(* append </Case> tag *)
					strString := '</Case>';
					nStringLen := LEN(strString);
					MEMMOVE(ADR(arrCACImage[nCACByte]), ADR(strString), nStringLen);
					nCACByte := nCACByte + nStringLen;

					eState := E_CAC_WRITEXMLIMAGE;
*)
				END_IF

			(* open file error *)
			ELSE

				bError := TRUE;
				nErrorID := fbOpenFile.nErrID;
				eErrorState := eState;

				eState := E_CAC_DONE;
			END_IF

			(* close off fbOpenFile *)
			fbOpenFile(bExecute := FALSE);
		END_IF


	(* build XML image for CAC data *)
	E_CAC_BUILDXMLIMAGE:

	(* Reset *)
		fbPopulateMinimalOuterData(
			bExecute := FALSE,
			nNumberofOuters := stCACData.NumberOfOuters,
			stCACData := stCACData
		);

